   1:  PR[GP1:91,1] = PR[GP1:90,1] + -29.809;
   1:  PR[GP1:91,2] = PR[GP1:90,2] + -36.321;
   1:L PR[91] 10mm/sec CNT100;
   1:  PR[GP1:91,1] = PR[GP1:90,1] + -23.100;
   1:  PR[GP1:91,2] = PR[GP1:90,2] + -35.878;
   1:L PR[91] 10mm/sec CNT100;
   1:  PR[GP1:91,1] = PR[GP1:90,1] + -20.028;
   1:  PR[GP1:91,2] = PR[GP1:90,2] + -35.175;
   1:L PR[91] 10mm/sec CNT100;
   1:  PR[GP1:91,1] = PR[GP1:90,1] + -13.814;
   1:  PR[GP1:91,2] = PR[GP1:90,2] + -33.391;
   1:L PR[91] 10mm/sec CNT100;
   1:  PR[GP1:91,1] = PR[GP1:90,1] + -10.898;
   1:  PR[GP1:91,2] = PR[GP1:90,2] + -31.682;
   1:L PR[91] 10mm/sec CNT100;
   1:  PR[GP1:91,1] = PR[GP1:90,1] + -6.741;
   1:  PR[GP1:91,2] = PR[GP1:90,2] + -29.419;
   1:L PR[91] 10mm/sec CNT100;
   1:  PR[GP1:91,1] = PR[GP1:90,1] + -1.126;
   1:  PR[GP1:91,2] = PR[GP1:90,2] + -24.565;
   1:L PR[91] 10mm/sec CNT100;
   1:  PR[GP1:91,1] = PR[GP1:90,1] + -0.604;
   1:  PR[GP1:91,2] = PR[GP1:90,2] + -23.932;
   1:L PR[91] 10mm/sec CNT100;
   1:  PR[GP1:91,1] = PR[GP1:90,1] + 0.084;
   1:L PR[91] 10mm/sec CNT100;
   1:  PR[GP1:91,1] = PR[GP1:90,1] + 0.382;
   1:  PR[GP1:91,2] = PR[GP1:90,2] + -24.658;
   1:  PR[GP1:91,3] = PR[GP1:90,3] + 53.375;
   1:L PR[91] 10mm/sec CNT100;
   1:  PR[GP1:91,1] = PR[GP1:90,1] + 0.577;
   1:  PR[GP1:91,2] = PR[GP1:90,2] + -24.830;
   1:L PR[91] 10mm/sec CNT100;
   1:  PR[GP1:91,1] = PR[GP1:90,1] + 5.985;
   1:  PR[GP1:91,2] = PR[GP1:90,2] + -29.504;
   1:L PR[91] 10mm/sec CNT100;
   1:  PR[GP1:91,1] = PR[GP1:90,1] + 9.953;
   1:  PR[GP1:91,2] = PR[GP1:90,2] + -31.657;
   1:L PR[91] 10mm/sec CNT100;
   1:  PR[GP1:91,1] = PR[GP1:90,1] + 13.028;
   1:  PR[GP1:91,2] = PR[GP1:90,2] + -33.457;
   1:L PR[91] 10mm/sec CNT100;
   1:  PR[GP1:91,1] = PR[GP1:90,1] + 19.129;
   1:  PR[GP1:91,2] = PR[GP1:90,2] + -35.209;
   1:L PR[91] 10mm/sec CNT100;
   1:  PR[GP1:91,1] = PR[GP1:90,1] + 22.400;
   1:  PR[GP1:91,2] = PR[GP1:90,2] + -35.958;
   1:L PR[91] 10mm/sec CNT100;
   1:  PR[GP1:91,1] = PR[GP1:90,1] + 28.952;
   1:  PR[GP1:91,2] = PR[GP1:90,2] + -36.393;
   1:L PR[91] 10mm/sec CNT100;
   1:  PR[GP1:91,1] = PR[GP1:90,1] + 36.269;
   1:  PR[GP1:91,2] = PR[GP1:90,2] + -35.383;
   1:L PR[91] 10mm/sec CNT100;
   1:  PR[GP1:91,1] = PR[GP1:90,1] + 38.372;
   1:  PR[GP1:91,2] = PR[GP1:90,2] + -35.179;
   1:L PR[91] 10mm/sec CNT100;
   1:  PR[GP1:91,1] = PR[GP1:90,1] + 45.492;
   1:  PR[GP1:91,2] = PR[GP1:90,2] + -32.580;
   1:L PR[91] 10mm/sec CNT100;
   1:  PR[GP1:91,1] = PR[GP1:90,1] + 46.753;
   1:  PR[GP1:91,2] = PR[GP1:90,2] + -32.025;
   1:L PR[91] 10mm/sec CNT100;
   1:  PR[GP1:91,1] = PR[GP1:90,1] + 53.239;
   1:  PR[GP1:91,2] = PR[GP1:90,2] + -27.956;
   1:L PR[91] 10mm/sec CNT100;
   1:  PR[GP1:91,1] = PR[GP1:90,1] + 59.284;
   1:  PR[GP1:91,2] = PR[GP1:90,2] + -22.078;
   1:L PR[91] 10mm/sec CNT100;
   1:  PR[GP1:91,1] = PR[GP1:90,1] + 62.332;
   1:  PR[GP1:91,2] = PR[GP1:90,2] + -17.349;
   1:L PR[91] 10mm/sec CNT100;
   1:  PR[GP1:91,1] = PR[GP1:90,1] + 63.823;
   1:  PR[GP1:91,2] = PR[GP1:90,2] + -15.009;
   1:L PR[91] 10mm/sec CNT100;
   1:  PR[GP1:91,1] = PR[GP1:90,1] + 66.412;
   1:  PR[GP1:91,2] = PR[GP1:90,2] + -8.017;
   1:L PR[91] 10mm/sec CNT100;
   1:  PR[GP1:91,1] = PR[GP1:90,1] + 66.615;
   1:  PR[GP1:91,2] = PR[GP1:90,2] + -6.897;
   1:L PR[91] 10mm/sec CNT100;
   1:  PR[GP1:91,1] = PR[GP1:90,1] + 67.423;
   1:  PR[GP1:91,2] = PR[GP1:90,2] + 0.258;
   1:L PR[91] 10mm/sec CNT100;
   1:  PR[GP1:91,1] = PR[GP1:90,1] + 67.185;
   1:  PR[GP1:91,2] = PR[GP1:90,2] + 1.554;
   1:L PR[91] 10mm/sec CNT100;
   1:  PR[GP1:91,1] = PR[GP1:90,1] + 66.405;
   1:  PR[GP1:91,2] = PR[GP1:90,2] + 8.595;
   1:L PR[91] 10mm/sec CNT100;
   1:  PR[GP1:91,1] = PR[GP1:90,1] + 63.820;
   1:  PR[GP1:91,2] = PR[GP1:90,2] + 15.577;
   1:L PR[91] 10mm/sec CNT100;
   1:  PR[GP1:91,1] = PR[GP1:90,1] + 63.649;
   1:  PR[GP1:91,2] = PR[GP1:90,2] + 15.865;
   1:L PR[91] 10mm/sec CNT100;
   1:  PR[GP1:91,1] = PR[GP1:90,1] + 59.282;
   1:  PR[GP1:91,2] = PR[GP1:90,2] + 22.638;
   1:L PR[91] 10mm/sec CNT100;
   1:  PR[GP1:91,1] = PR[GP1:90,1] + 53.786;
   1:  PR[GP1:91,2] = PR[GP1:90,2] + 28.020;
   1:L PR[91] 10mm/sec CNT100;
   1:  PR[GP1:91,1] = PR[GP1:90,1] + 53.244;
   1:  PR[GP1:91,2] = PR[GP1:90,2] + 28.511;
   1:L PR[91] 10mm/sec CNT100;
   1:  PR[GP1:91,1] = PR[GP1:90,1] + 46.747;
   1:  PR[GP1:91,2] = PR[GP1:90,2] + 32.588;
   1:L PR[91] 10mm/sec CNT100;
   1:  PR[GP1:91,1] = PR[GP1:90,1] + 45.480;
   1:  PR[GP1:91,2] = PR[GP1:90,2] + 33.141;
   1:L PR[91] 10mm/sec CNT100;
   1:  PR[GP1:91,1] = PR[GP1:90,1] + 38.342;
   1:  PR[GP1:91,2] = PR[GP1:90,2] + 35.746;
   1:L PR[91] 10mm/sec CNT100;
   1:  PR[GP1:91,1] = PR[GP1:90,1] + 31.583;
   1:  PR[GP1:91,2] = PR[GP1:90,2] + 36.704;
   1:L PR[91] 10mm/sec CNT100;
   1:  PR[GP1:91,1] = PR[GP1:90,1] + 28.935;
   1:  PR[GP1:91,2] = PR[GP1:90,2] + 36.950;
   1:L PR[91] 10mm/sec CNT100;
   1:  PR[GP1:91,1] = PR[GP1:90,1] + 22.366;
   1:  PR[GP1:91,2] = PR[GP1:90,2] + 36.514;
   1:L PR[91] 10mm/sec CNT100;
   1:  PR[GP1:91,1] = PR[GP1:90,1] + 19.041;
   1:  PR[GP1:91,2] = PR[GP1:90,2] + 35.728;
   1:L PR[91] 10mm/sec CNT100;
   1:  PR[GP1:91,1] = PR[GP1:90,1] + 12.948;
   1:  PR[GP1:91,2] = PR[GP1:90,2] + 33.976;
   1:L PR[91] 10mm/sec CNT100;
   1:  PR[GP1:91,1] = PR[GP1:90,1] + 7.626;
   1:  PR[GP1:91,2] = PR[GP1:90,2] + 31.111;
   1:L PR[91] 10mm/sec CNT100;
   1:  PR[GP1:91,1] = PR[GP1:90,1] + 0.493;
   1:  PR[GP1:91,2] = PR[GP1:90,2] + 25.310;
   1:L PR[91] 10mm/sec CNT100;
   1:  PR[GP1:91,1] = PR[GP1:90,1] + 0.344;
   1:  PR[GP1:91,2] = PR[GP1:90,2] + 25.179;
   1:L PR[91] 10mm/sec CNT100;
   1:  PR[GP1:91,1] = PR[GP1:90,1] + 0.046;
   1:  PR[GP1:91,2] = PR[GP1:90,2] + 24.815;
   1:L PR[91] 10mm/sec CNT100;
   1:  PR[GP1:91,1] = PR[GP1:90,1] + -0.570;
   1:L PR[91] 10mm/sec CNT100;
   1:  PR[GP1:91,1] = PR[GP1:90,1] + -0.868;
   1:  PR[GP1:91,2] = PR[GP1:90,2] + 25.177;
   1:L PR[91] 10mm/sec CNT100;
   1:  PR[GP1:91,1] = PR[GP1:90,1] + -1.018;
   1:  PR[GP1:91,2] = PR[GP1:90,2] + 25.309;
   1:L PR[91] 10mm/sec CNT100;
   1:  PR[GP1:91,1] = PR[GP1:90,1] + -8.130;
   1:  PR[GP1:91,2] = PR[GP1:90,2] + 31.091;
   1:L PR[91] 10mm/sec CNT100;
   1:  PR[GP1:91,1] = PR[GP1:90,1] + -13.479;
   1:  PR[GP1:91,2] = PR[GP1:90,2] + 33.979;
   1:L PR[91] 10mm/sec CNT100;
   1:  PR[GP1:91,1] = PR[GP1:90,1] + -19.564;
   1:  PR[GP1:91,2] = PR[GP1:90,2] + 35.729;
   1:L PR[91] 10mm/sec CNT100;
   1:  PR[GP1:91,1] = PR[GP1:90,1] + -22.890;
   1:  PR[GP1:91,2] = PR[GP1:90,2] + 36.514;
   1:L PR[91] 10mm/sec CNT100;
   1:  PR[GP1:91,1] = PR[GP1:90,1] + -29.466;
   1:  PR[GP1:91,2] = PR[GP1:90,2] + 36.948;
   1:L PR[91] 10mm/sec CNT100;
   1:  PR[GP1:91,1] = PR[GP1:90,1] + -36.812;
   1:  PR[GP1:91,2] = PR[GP1:90,2] + 35.931;
   1:L PR[91] 10mm/sec CNT100;
   1:  PR[GP1:91,1] = PR[GP1:90,1] + -38.919;
   1:  PR[GP1:91,2] = PR[GP1:90,2] + 35.733;
   1:L PR[91] 10mm/sec CNT100;
   1:  PR[GP1:91,1] = PR[GP1:90,1] + -46.035;
   1:  PR[GP1:91,2] = PR[GP1:90,2] + 33.127;
   1:L PR[91] 10mm/sec CNT100;
   1:  PR[GP1:91,1] = PR[GP1:90,1] + -47.299;
   1:  PR[GP1:91,2] = PR[GP1:90,2] + 32.574;
   1:L PR[91] 10mm/sec CNT100;
   1:  PR[GP1:91,1] = PR[GP1:90,1] + -53.827;
   1:  PR[GP1:91,2] = PR[GP1:90,2] + 28.459;
   1:L PR[91] 10mm/sec CNT100;
   1:  PR[GP1:91,1] = PR[GP1:90,1] + -59.727;
   1:  PR[GP1:91,2] = PR[GP1:90,2] + 22.699;
   1:L PR[91] 10mm/sec CNT100;
   1:  PR[GP1:91,1] = PR[GP1:90,1] + -59.886;
   1:  PR[GP1:91,2] = PR[GP1:90,2] + 22.555;
   1:L PR[91] 10mm/sec CNT100;
   1:  PR[GP1:91,1] = PR[GP1:90,1] + -62.857;
   1:  PR[GP1:91,2] = PR[GP1:90,2] + 17.918;
   1:L PR[91] 10mm/sec CNT100;
   1:  PR[GP1:91,1] = PR[GP1:90,1] + -64.370;
   1:  PR[GP1:91,2] = PR[GP1:90,2] + 15.527;
   1:L PR[91] 10mm/sec CNT100;
   1:  PR[GP1:91,1] = PR[GP1:90,1] + -66.967;
   1:  PR[GP1:91,2] = PR[GP1:90,2] + 8.422;
   1:L PR[91] 10mm/sec CNT100;
   1:  PR[GP1:91,1] = PR[GP1:90,1] + -67.171;
   1:  PR[GP1:91,2] = PR[GP1:90,2] + 7.296;
   1:L PR[91] 10mm/sec CNT100;
   1:  PR[GP1:91,1] = PR[GP1:90,1] + -67.949;
   1:  PR[GP1:91,2] = PR[GP1:90,2] + 0.301;
   1:L PR[91] 10mm/sec CNT100;
   1:  PR[GP1:91,1] = PR[GP1:90,1] + -67.711;
   1:  PR[GP1:91,2] = PR[GP1:90,2] + -0.994;
   1:L PR[91] 10mm/sec CNT100;
   1:  PR[GP1:91,1] = PR[GP1:90,1] + -66.959;
   1:  PR[GP1:91,2] = PR[GP1:90,2] + -7.884;
   1:L PR[91] 10mm/sec CNT100;
   1:  PR[GP1:91,1] = PR[GP1:90,1] + -64.367;
   1:  PR[GP1:91,2] = PR[GP1:90,2] + -14.977;
   1:L PR[91] 10mm/sec CNT100;
   1:  PR[GP1:91,1] = PR[GP1:90,1] + -64.194;
   1:  PR[GP1:91,2] = PR[GP1:90,2] + -15.271;
   1:L PR[91] 10mm/sec CNT100;
   1:  PR[GP1:91,1] = PR[GP1:90,1] + -59.880;
   1:  PR[GP1:91,2] = PR[GP1:90,2] + -22.006;
   1:L PR[91] 10mm/sec CNT100;
   1:  PR[GP1:91,1] = PR[GP1:90,1] + -54.377;
   1:  PR[GP1:91,2] = PR[GP1:90,2] + -27.405;
   1:L PR[91] 10mm/sec CNT100;
   1:  PR[GP1:91,1] = PR[GP1:90,1] + -53.841;
   1:  PR[GP1:91,2] = PR[GP1:90,2] + -27.892;
   1:L PR[91] 10mm/sec CNT100;
   1:  PR[GP1:91,1] = PR[GP1:90,1] + -47.306;
   1:  PR[GP1:91,2] = PR[GP1:90,2] + -32.012;
   1:L PR[91] 10mm/sec CNT100;
   1:  PR[GP1:91,1] = PR[GP1:90,1] + -46.047;
   1:  PR[GP1:91,2] = PR[GP1:90,2] + -32.566;
   1:L PR[91] 10mm/sec CNT100;
   1:  PR[GP1:91,1] = PR[GP1:90,1] + -38.923;
   1:  PR[GP1:91,2] = PR[GP1:90,2] + -35.176;
   1:L PR[91] 10mm/sec CNT100;
   1:  PR[GP1:91,1] = PR[GP1:90,1] + -32.147;
   1:  PR[GP1:91,2] = PR[GP1:90,2] + -36.140;
   1:L PR[91] 10mm/sec CNT100;
   1:  PR[GP1:91,1] = PR[GP1:90,1] + -29.509;
   1:  PR[GP1:91,2] = PR[GP1:90,2] + -36.393;
   1:L PR[91] 10mm/sec CNT100;
   1:  PR[GP1:91,1] = PR[GP1:90,1] + -22.924;
   1:  PR[GP1:91,2] = PR[GP1:90,2] + -35.958;
   1:L PR[91] 10mm/sec CNT100;
   1:  PR[GP1:91,1] = PR[GP1:90,1] + -19.653;
   1:  PR[GP1:91,2] = PR[GP1:90,2] + -35.210;
   1:L PR[91] 10mm/sec CNT100;
   1:  PR[GP1:91,1] = PR[GP1:90,1] + -13.560;
   1:  PR[GP1:91,2] = PR[GP1:90,2] + -33.460;
   1:L PR[91] 10mm/sec CNT100;
   1:  PR[GP1:91,1] = PR[GP1:90,1] + -10.487;
   1:  PR[GP1:91,2] = PR[GP1:90,2] + -31.660;
   1:L PR[91] 10mm/sec CNT100;
   1:  PR[GP1:91,1] = PR[GP1:90,1] + -6.497;
   1:  PR[GP1:91,2] = PR[GP1:90,2] + -29.488;
   1:L PR[91] 10mm/sec CNT100;
   1:  PR[GP1:91,1] = PR[GP1:90,1] + -1.098;
   1:  PR[GP1:91,2] = PR[GP1:90,2] + -24.829;
   1:L PR[91] 10mm/sec CNT100;
   1:  PR[GP1:91,1] = PR[GP1:90,1] + -0.902;
   1:  PR[GP1:91,2] = PR[GP1:90,2] + -24.656;
   1:L PR[91] 10mm/sec CNT100;
   1:  PR[GP1:91,1] = PR[GP1:90,1] + -0.573;
   1:  PR[GP1:91,2] = PR[GP1:90,2] + -24.257;
   1:L PR[91] 10mm/sec CNT100;
   1:  PR[GP1:91,1] = PR[GP1:90,1] + 0.052;
   1:L PR[91] 10mm/sec CNT100;
   1:  PR[GP1:91,1] = PR[GP1:90,1] + 5.741;
   1:  PR[GP1:91,2] = PR[GP1:90,2] + -29.572;
   1:  PR[GP1:91,3] = PR[GP1:90,3] + 53.985;
   1:L PR[91] 10mm/sec CNT100;
   1:  PR[GP1:91,1] = PR[GP1:90,1] + 9.542;
   1:  PR[GP1:91,2] = PR[GP1:90,2] + -31.635;
   1:L PR[91] 10mm/sec CNT100;
   1:  PR[GP1:91,1] = PR[GP1:90,1] + 12.773;
   1:  PR[GP1:91,2] = PR[GP1:90,2] + -33.526;
   1:L PR[91] 10mm/sec CNT100;
   1:  PR[GP1:91,1] = PR[GP1:90,1] + 18.753;
   1:  PR[GP1:91,2] = PR[GP1:90,2] + -35.244;
   1:L PR[91] 10mm/sec CNT100;
   1:  PR[GP1:91,1] = PR[GP1:90,1] + 22.223;
   1:  PR[GP1:91,2] = PR[GP1:90,2] + -36.038;
   1:L PR[91] 10mm/sec CNT100;
   1:  PR[GP1:91,1] = PR[GP1:90,1] + 28.652;
   1:  PR[GP1:91,2] = PR[GP1:90,2] + -36.465;
   1:L PR[91] 10mm/sec CNT100;
   1:  PR[GP1:91,1] = PR[GP1:90,1] + 35.832;
   1:  PR[GP1:91,2] = PR[GP1:90,2] + -35.474;
   1:L PR[91] 10mm/sec CNT100;
   1:  PR[GP1:91,1] = PR[GP1:90,1] + 38.154;
   1:  PR[GP1:91,2] = PR[GP1:90,2] + -35.248;
   1:L PR[91] 10mm/sec CNT100;
   1:  PR[GP1:91,1] = PR[GP1:90,1] + 45.148;
   1:  PR[GP1:91,2] = PR[GP1:90,2] + -32.696;
   1:L PR[91] 10mm/sec CNT100;
   1:  PR[GP1:91,1] = PR[GP1:90,1] + 46.608;
   1:  PR[GP1:91,2] = PR[GP1:90,2] + -32.053;
   1:L PR[91] 10mm/sec CNT100;
   1:  PR[GP1:91,1] = PR[GP1:90,1] + 52.984;
   1:  PR[GP1:91,2] = PR[GP1:90,2] + -28.053;
   1:L PR[91] 10mm/sec CNT100;
   1:  PR[GP1:91,1] = PR[GP1:90,1] + 58.770;
   1:  PR[GP1:91,2] = PR[GP1:90,2] + -22.413;
   1:L PR[91] 10mm/sec CNT100;
   1:  PR[GP1:91,1] = PR[GP1:90,1] + 59.102;
   1:  PR[GP1:91,2] = PR[GP1:90,2] + -22.111;
   1:L PR[91] 10mm/sec CNT100;
   1:  PR[GP1:91,1] = PR[GP1:90,1] + 63.606;
   1:  PR[GP1:91,2] = PR[GP1:90,2] + -15.115;
   1:L PR[91] 10mm/sec CNT100;
   1:  PR[GP1:91,1] = PR[GP1:90,1] + 66.309;
   1:  PR[GP1:91,2] = PR[GP1:90,2] + -7.800;
   1:L PR[91] 10mm/sec CNT100;
   1:  PR[GP1:91,1] = PR[GP1:90,1] + 66.390;
   1:  PR[GP1:91,2] = PR[GP1:90,2] + -7.350;
   1:L PR[91] 10mm/sec CNT100;
   1:  PR[GP1:91,1] = PR[GP1:90,1] + 67.249;
   1:  PR[GP1:91,2] = PR[GP1:90,2] + 0.258;
   1:L PR[91] 10mm/sec CNT100;
   1:  PR[GP1:91,1] = PR[GP1:90,1] + 67.127;
   1:  PR[GP1:91,2] = PR[GP1:90,2] + 0.921;
   1:L PR[91] 10mm/sec CNT100;
   1:  PR[GP1:91,1] = PR[GP1:90,1] + 66.301;
   1:  PR[GP1:91,2] = PR[GP1:90,2] + 8.377;
   1:L PR[91] 10mm/sec CNT100;
   1:  PR[GP1:91,1] = PR[GP1:90,1] + 63.606;
   1:  PR[GP1:91,2] = PR[GP1:90,2] + 15.673;
   1:L PR[91] 10mm/sec CNT100;
   1:  PR[GP1:91,1] = PR[GP1:90,1] + 59.095;
   1:  PR[GP1:91,2] = PR[GP1:90,2] + 22.680;
   1:L PR[91] 10mm/sec CNT100;
   1:  PR[GP1:91,1] = PR[GP1:90,1] + 53.689;
   1:  PR[GP1:91,2] = PR[GP1:90,2] + 27.974;
   1:L PR[91] 10mm/sec CNT100;
   1:  PR[GP1:91,1] = PR[GP1:90,1] + 52.987;
   1:  PR[GP1:91,2] = PR[GP1:90,2] + 28.609;
   1:L PR[91] 10mm/sec CNT100;
   1:  PR[GP1:91,1] = PR[GP1:90,1] + 46.600;
   1:  PR[GP1:91,2] = PR[GP1:90,2] + 32.617;
   1:L PR[91] 10mm/sec CNT100;
   1:  PR[GP1:91,1] = PR[GP1:90,1] + 45.134;
   1:  PR[GP1:91,2] = PR[GP1:90,2] + 33.257;
   1:L PR[91] 10mm/sec CNT100;
   1:  PR[GP1:91,1] = PR[GP1:90,1] + 38.123;
   1:  PR[GP1:91,2] = PR[GP1:90,2] + 35.816;
   1:L PR[91] 10mm/sec CNT100;
   1:  PR[GP1:91,1] = PR[GP1:90,1] + 31.484;
   1:  PR[GP1:91,2] = PR[GP1:90,2] + 36.757;
   1:L PR[91] 10mm/sec CNT100;
   1:  PR[GP1:91,1] = PR[GP1:90,1] + 28.633;
   1:  PR[GP1:91,2] = PR[GP1:90,2] + 37.022;
   1:L PR[91] 10mm/sec CNT100;
   1:  PR[GP1:91,1] = PR[GP1:90,1] + 22.187;
   1:  PR[GP1:91,2] = PR[GP1:90,2] + 36.594;
   1:L PR[91] 10mm/sec CNT100;
   1:  PR[GP1:91,1] = PR[GP1:90,1] + 18.660;
   1:  PR[GP1:91,2] = PR[GP1:90,2] + 35.761;
   1:L PR[91] 10mm/sec CNT100;
   1:  PR[GP1:91,1] = PR[GP1:90,1] + 12.690;
   1:  PR[GP1:91,2] = PR[GP1:90,2] + 34.044;
   1:L PR[91] 10mm/sec CNT100;
   1:  PR[GP1:91,1] = PR[GP1:90,1] + 7.453;
   1:  PR[GP1:91,2] = PR[GP1:90,2] + 31.225;
   1:L PR[91] 10mm/sec CNT100;
   1:  PR[GP1:91,1] = PR[GP1:90,1] + -0.263;
   1:  PR[GP1:91,2] = PR[GP1:90,2] + 24.950;
   1:L PR[91] 10mm/sec CNT100;
   1:  PR[GP1:91,1] = PR[GP1:90,1] + -7.958;
   1:  PR[GP1:91,2] = PR[GP1:90,2] + 31.206;
   1:L PR[91] 10mm/sec CNT100;
   1:  PR[GP1:91,1] = PR[GP1:90,1] + -13.221;
   1:  PR[GP1:91,2] = PR[GP1:90,2] + 34.047;
   1:L PR[91] 10mm/sec CNT100;
   1:  PR[GP1:91,1] = PR[GP1:90,1] + -19.183;
   1:  PR[GP1:91,2] = PR[GP1:90,2] + 35.761;
   1:L PR[91] 10mm/sec CNT100;
   1:  PR[GP1:91,1] = PR[GP1:90,1] + -22.711;
   1:  PR[GP1:91,2] = PR[GP1:90,2] + 36.594;
   1:L PR[91] 10mm/sec CNT100;
   1:  PR[GP1:91,1] = PR[GP1:90,1] + -29.163;
   1:  PR[GP1:91,2] = PR[GP1:90,2] + 37.020;
   1:L PR[91] 10mm/sec CNT100;
   1:  PR[GP1:91,1] = PR[GP1:90,1] + -36.373;
   1:  PR[GP1:91,2] = PR[GP1:90,2] + 36.022;
   1:L PR[91] 10mm/sec CNT100;
   1:  PR[GP1:91,1] = PR[GP1:90,1] + -38.699;
   1:  PR[GP1:91,2] = PR[GP1:90,2] + 35.803;
   1:L PR[91] 10mm/sec CNT100;
   1:  PR[GP1:91,1] = PR[GP1:90,1] + -45.689;
   1:  PR[GP1:91,2] = PR[GP1:90,2] + 33.243;
   1:L PR[91] 10mm/sec CNT100;
   1:  PR[GP1:91,1] = PR[GP1:90,1] + -47.153;
   1:  PR[GP1:91,2] = PR[GP1:90,2] + 32.603;
   1:L PR[91] 10mm/sec CNT100;
   1:  PR[GP1:91,1] = PR[GP1:90,1] + -53.569;
   1:  PR[GP1:91,2] = PR[GP1:90,2] + 28.558;
   1:L PR[91] 10mm/sec CNT100;
   1:  PR[GP1:91,1] = PR[GP1:90,1] + -59.370;
   1:  PR[GP1:91,2] = PR[GP1:90,2] + 22.895;
   1:L PR[91] 10mm/sec CNT100;
   1:  PR[GP1:91,1] = PR[GP1:90,1] + -59.698;
   1:  PR[GP1:91,2] = PR[GP1:90,2] + 22.598;
   1:L PR[91] 10mm/sec CNT100;
   1:  PR[GP1:91,1] = PR[GP1:90,1] + -64.153;
   1:  PR[GP1:91,2] = PR[GP1:90,2] + 15.634;
   1:L PR[91] 10mm/sec CNT100;
   1:  PR[GP1:91,1] = PR[GP1:90,1] + -66.865;
   1:  PR[GP1:91,2] = PR[GP1:90,2] + 8.197;
   1:L PR[91] 10mm/sec CNT100;
   1:  PR[GP1:91,1] = PR[GP1:90,1] + -66.948;
   1:  PR[GP1:91,2] = PR[GP1:90,2] + 7.740;
   1:L PR[91] 10mm/sec CNT100;
   1:  PR[GP1:91,1] = PR[GP1:90,1] + -67.775;
   1:  PR[GP1:91,2] = PR[GP1:90,2] + 0.301;
   1:L PR[91] 10mm/sec CNT100;
   1:  PR[GP1:91,1] = PR[GP1:90,1] + -67.653;
   1:  PR[GP1:91,2] = PR[GP1:90,2] + -0.362;
   1:L PR[91] 10mm/sec CNT100;
   1:  PR[GP1:91,1] = PR[GP1:90,1] + -66.857;
   1:  PR[GP1:91,2] = PR[GP1:90,2] + -7.659;
   1:L PR[91] 10mm/sec CNT100;
   1:  PR[GP1:91,1] = PR[GP1:90,1] + -64.146;
   1:  PR[GP1:91,2] = PR[GP1:90,2] + -15.094;
   1:L PR[91] 10mm/sec CNT100;
   1:  PR[GP1:91,1] = PR[GP1:90,1] + -64.138;
   1:  PR[GP1:91,2] = PR[GP1:90,2] + -15.110;
   1:L PR[91] 10mm/sec CNT100;
   1:  PR[GP1:91,1] = PR[GP1:90,1] + -59.692;
   1:  PR[GP1:91,2] = PR[GP1:90,2] + -22.049;
   1:L PR[91] 10mm/sec CNT100;
   1:  PR[GP1:91,1] = PR[GP1:90,1] + -54.279;
   1:  PR[GP1:91,2] = PR[GP1:90,2] + -27.360;
   1:L PR[91] 10mm/sec CNT100;
   1:  PR[GP1:91,1] = PR[GP1:90,1] + -53.584;
   1:  PR[GP1:91,2] = PR[GP1:90,2] + -27.990;
   1:L PR[91] 10mm/sec CNT100;
   1:  PR[GP1:91,1] = PR[GP1:90,1] + -47.161;
   1:  PR[GP1:91,2] = PR[GP1:90,2] + -32.040;
   1:L PR[91] 10mm/sec CNT100;
   1:  PR[GP1:91,1] = PR[GP1:90,1] + -45.703;
   1:  PR[GP1:91,2] = PR[GP1:90,2] + -32.682;
   1:L PR[91] 10mm/sec CNT100;
   1:  PR[GP1:91,1] = PR[GP1:90,1] + -38.705;
   1:  PR[GP1:91,2] = PR[GP1:90,2] + -35.245;
   1:L PR[91] 10mm/sec CNT100;
   1:  PR[GP1:91,1] = PR[GP1:90,1] + -32.049;
   1:  PR[GP1:91,2] = PR[GP1:90,2] + -36.192;
   1:L PR[91] 10mm/sec CNT100;
   1:  PR[GP1:91,1] = PR[GP1:90,1] + -29.209;
   1:  PR[GP1:91,2] = PR[GP1:90,2] + -36.465;
   1:L PR[91] 10mm/sec CNT100;
   1:  PR[GP1:91,1] = PR[GP1:90,1] + -22.747;
   1:  PR[GP1:91,2] = PR[GP1:90,2] + -36.038;
   1:L PR[91] 10mm/sec CNT100;
   1:  PR[GP1:91,1] = PR[GP1:90,1] + -19.277;
   1:  PR[GP1:91,2] = PR[GP1:90,2] + -35.245;
   1:L PR[91] 10mm/sec CNT100;
   1:  PR[GP1:91,1] = PR[GP1:90,1] + -13.305;
   1:  PR[GP1:91,2] = PR[GP1:90,2] + -33.529;
   1:L PR[91] 10mm/sec CNT100;
   1:  PR[GP1:91,1] = PR[GP1:90,1] + -10.076;
   1:  PR[GP1:91,2] = PR[GP1:90,2] + -31.638;
   1:L PR[91] 10mm/sec CNT100;
   1:  PR[GP1:91,1] = PR[GP1:90,1] + -6.254;
   1:  PR[GP1:91,2] = PR[GP1:90,2] + -29.557;
   1:L PR[91] 10mm/sec CNT100;
   1:  PR[GP1:91,1] = PR[GP1:90,1] + -0.261;
   1:  PR[GP1:91,2] = PR[GP1:90,2] + -24.385;
   1:L PR[91] 10mm/sec CNT100;
   1:  PR[GP1:91,1] = PR[GP1:90,1] + 5.496;
   1:  PR[GP1:91,2] = PR[GP1:90,2] + -29.641;
   1:  PR[GP1:91,3] = PR[GP1:90,3] + 54.595;
   1:L PR[91] 10mm/sec CNT100;
   1:  PR[GP1:91,1] = PR[GP1:90,1] + 9.132;
   1:  PR[GP1:91,2] = PR[GP1:90,2] + -31.614;
   1:L PR[91] 10mm/sec CNT100;
   1:  PR[GP1:91,1] = PR[GP1:90,1] + 12.518;
   1:  PR[GP1:91,2] = PR[GP1:90,2] + -33.596;
   1:L PR[91] 10mm/sec CNT100;
   1:  PR[GP1:91,1] = PR[GP1:90,1] + 18.378;
   1:  PR[GP1:91,2] = PR[GP1:90,2] + -35.279;
   1:L PR[91] 10mm/sec CNT100;
   1:  PR[GP1:91,1] = PR[GP1:90,1] + 22.046;
   1:  PR[GP1:91,2] = PR[GP1:90,2] + -36.118;
   1:L PR[91] 10mm/sec CNT100;
   1:  PR[GP1:91,1] = PR[GP1:90,1] + 28.352;
   1:  PR[GP1:91,2] = PR[GP1:90,2] + -36.537;
   1:L PR[91] 10mm/sec CNT100;
   1:  PR[GP1:91,1] = PR[GP1:90,1] + 35.396;
   1:  PR[GP1:91,2] = PR[GP1:90,2] + -35.565;
   1:L PR[91] 10mm/sec CNT100;
   1:  PR[GP1:91,1] = PR[GP1:90,1] + 37.937;
   1:  PR[GP1:91,2] = PR[GP1:90,2] + -35.318;
   1:L PR[91] 10mm/sec CNT100;
   1:  PR[GP1:91,1] = PR[GP1:90,1] + 44.804;
   1:  PR[GP1:91,2] = PR[GP1:90,2] + -32.811;
   1:L PR[91] 10mm/sec CNT100;
   1:  PR[GP1:91,1] = PR[GP1:90,1] + 46.463;
   1:  PR[GP1:91,2] = PR[GP1:90,2] + -32.082;
   1:L PR[91] 10mm/sec CNT100;
   1:  PR[GP1:91,1] = PR[GP1:90,1] + 52.728;
   1:  PR[GP1:91,2] = PR[GP1:90,2] + -28.151;
   1:L PR[91] 10mm/sec CNT100;
   1:  PR[GP1:91,1] = PR[GP1:90,1] + 58.415;
   1:  PR[GP1:91,2] = PR[GP1:90,2] + -22.607;
   1:L PR[91] 10mm/sec CNT100;
   1:  PR[GP1:91,1] = PR[GP1:90,1] + 58.915;
   1:  PR[GP1:91,2] = PR[GP1:90,2] + -22.153;
   1:L PR[91] 10mm/sec CNT100;
   1:  PR[GP1:91,1] = PR[GP1:90,1] + 63.327;
   1:  PR[GP1:91,2] = PR[GP1:90,2] + -15.309;
   1:L PR[91] 10mm/sec CNT100;
   1:  PR[GP1:91,1] = PR[GP1:90,1] + 63.445;
   1:  PR[GP1:91,2] = PR[GP1:90,2] + -15.097;
   1:L PR[91] 10mm/sec CNT100;
   1:  PR[GP1:91,1] = PR[GP1:90,1] + 66.176;
   1:  PR[GP1:91,2] = PR[GP1:90,2] + -7.670;
   1:L PR[91] 10mm/sec CNT100;
   1:  PR[GP1:91,1] = PR[GP1:90,1] + 67.077;
   1:  PR[GP1:91,2] = PR[GP1:90,2] + 0.279;
   1:L PR[91] 10mm/sec CNT100;
   1:  PR[GP1:91,1] = PR[GP1:90,1] + 66.176;
   1:  PR[GP1:91,2] = PR[GP1:90,2] + 8.228;
   1:L PR[91] 10mm/sec CNT100;
   1:  PR[GP1:91,1] = PR[GP1:90,1] + 63.445;
   1:  PR[GP1:91,2] = PR[GP1:90,2] + 15.656;
   1:L PR[91] 10mm/sec CNT100;
   1:  PR[GP1:91,1] = PR[GP1:90,1] + 63.327;
   1:  PR[GP1:91,2] = PR[GP1:90,2] + 15.868;
   1:L PR[91] 10mm/sec CNT100;
   1:  PR[GP1:91,1] = PR[GP1:90,1] + 58.907;
   1:  PR[GP1:91,2] = PR[GP1:90,2] + 22.722;
   1:L PR[91] 10mm/sec CNT100;
   1:  PR[GP1:91,1] = PR[GP1:90,1] + 53.591;
   1:  PR[GP1:91,2] = PR[GP1:90,2] + 27.928;
   1:L PR[91] 10mm/sec CNT100;
   1:  PR[GP1:91,1] = PR[GP1:90,1] + 52.731;
   1:  PR[GP1:91,2] = PR[GP1:90,2] + 28.707;
   1:L PR[91] 10mm/sec CNT100;
   1:  PR[GP1:91,1] = PR[GP1:90,1] + 46.454;
   1:  PR[GP1:91,2] = PR[GP1:90,2] + 32.646;
   1:L PR[91] 10mm/sec CNT100;
   1:  PR[GP1:91,1] = PR[GP1:90,1] + 44.788;
   1:  PR[GP1:91,2] = PR[GP1:90,2] + 33.373;
   1:L PR[91] 10mm/sec CNT100;
   1:  PR[GP1:91,1] = PR[GP1:90,1] + 37.903;
   1:  PR[GP1:91,2] = PR[GP1:90,2] + 35.886;
   1:L PR[91] 10mm/sec CNT100;
   1:  PR[GP1:91,1] = PR[GP1:90,1] + 31.385;
   1:  PR[GP1:91,2] = PR[GP1:90,2] + 36.810;
   1:L PR[91] 10mm/sec CNT100;
   1:  PR[GP1:91,1] = PR[GP1:90,1] + 28.331;
   1:  PR[GP1:91,2] = PR[GP1:90,2] + 37.094;
   1:L PR[91] 10mm/sec CNT100;
   1:  PR[GP1:91,1] = PR[GP1:90,1] + 22.009;
   1:  PR[GP1:91,2] = PR[GP1:90,2] + 36.674;
   1:L PR[91] 10mm/sec CNT100;
   1:  PR[GP1:91,1] = PR[GP1:90,1] + 18.280;
   1:  PR[GP1:91,2] = PR[GP1:90,2] + 35.793;
   1:L PR[91] 10mm/sec CNT100;
   1:  PR[GP1:91,1] = PR[GP1:90,1] + 12.432;
   1:  PR[GP1:91,2] = PR[GP1:90,2] + 34.112;
   1:L PR[91] 10mm/sec CNT100;
   1:  PR[GP1:91,1] = PR[GP1:90,1] + 7.280;
   1:  PR[GP1:91,2] = PR[GP1:90,2] + 31.339;
   1:L PR[91] 10mm/sec CNT100;
   1:  PR[GP1:91,1] = PR[GP1:90,1] + -0.263;
   1:  PR[GP1:91,2] = PR[GP1:90,2] + 25.204;
   1:L PR[91] 10mm/sec CNT100;
   1:  PR[GP1:91,1] = PR[GP1:90,1] + -7.786;
   1:  PR[GP1:91,2] = PR[GP1:90,2] + 31.321;
   1:L PR[91] 10mm/sec CNT100;
   1:  PR[GP1:91,1] = PR[GP1:90,1] + -12.962;
   1:  PR[GP1:91,2] = PR[GP1:90,2] + 34.115;
   1:L PR[91] 10mm/sec CNT100;
   1:  PR[GP1:91,1] = PR[GP1:90,1] + -18.802;
   1:  PR[GP1:91,2] = PR[GP1:90,2] + 35.794;
   1:L PR[91] 10mm/sec CNT100;
   1:  PR[GP1:91,1] = PR[GP1:90,1] + -22.532;
   1:  PR[GP1:91,2] = PR[GP1:90,2] + 36.674;
   1:L PR[91] 10mm/sec CNT100;
   1:  PR[GP1:91,1] = PR[GP1:90,1] + -28.861;
   1:  PR[GP1:91,2] = PR[GP1:90,2] + 37.092;
   1:L PR[91] 10mm/sec CNT100;
   1:  PR[GP1:91,1] = PR[GP1:90,1] + -35.934;
   1:  PR[GP1:91,2] = PR[GP1:90,2] + 36.113;
   1:L PR[91] 10mm/sec CNT100;
   1:  PR[GP1:91,1] = PR[GP1:90,1] + -38.479;
   1:  PR[GP1:91,2] = PR[GP1:90,2] + 35.874;
   1:L PR[91] 10mm/sec CNT100;
   1:  PR[GP1:91,1] = PR[GP1:90,1] + -45.342;
   1:  PR[GP1:91,2] = PR[GP1:90,2] + 33.360;
   1:L PR[91] 10mm/sec CNT100;
   1:  PR[GP1:91,1] = PR[GP1:90,1] + -47.006;
   1:  PR[GP1:91,2] = PR[GP1:90,2] + 32.633;
   1:L PR[91] 10mm/sec CNT100;
   1:  PR[GP1:91,1] = PR[GP1:90,1] + -53.311;
   1:  PR[GP1:91,2] = PR[GP1:90,2] + 28.657;
   1:L PR[91] 10mm/sec CNT100;
   1:  PR[GP1:91,1] = PR[GP1:90,1] + -59.012;
   1:  PR[GP1:91,2] = PR[GP1:90,2] + 23.092;
   1:L PR[91] 10mm/sec CNT100;
   1:  PR[GP1:91,1] = PR[GP1:90,1] + -59.509;
   1:  PR[GP1:91,2] = PR[GP1:90,2] + 22.642;
   1:L PR[91] 10mm/sec CNT100;
   1:  PR[GP1:91,1] = PR[GP1:90,1] + -63.875;
   1:  PR[GP1:91,2] = PR[GP1:90,2] + 15.828;
   1:L PR[91] 10mm/sec CNT100;
   1:  PR[GP1:91,1] = PR[GP1:90,1] + -63.992;
   1:  PR[GP1:91,2] = PR[GP1:90,2] + 15.617;
   1:L PR[91] 10mm/sec CNT100;
   1:  PR[GP1:91,1] = PR[GP1:90,1] + -66.735;
   1:  PR[GP1:91,2] = PR[GP1:90,2] + 8.058;
   1:L PR[91] 10mm/sec CNT100;
   1:  PR[GP1:91,1] = PR[GP1:90,1] + -67.601;
   1:  PR[GP1:91,2] = PR[GP1:90,2] + 0.301;
   1:L PR[91] 10mm/sec CNT100;
   1:  PR[GP1:91,1] = PR[GP1:90,1] + -67.596;
   1:  PR[GP1:91,2] = PR[GP1:90,2] + 0.270;
   1:L PR[91] 10mm/sec CNT100;
   1:  PR[GP1:91,1] = PR[GP1:90,1] + -66.735;
   1:  PR[GP1:91,2] = PR[GP1:90,2] + -7.500;
   1:L PR[91] 10mm/sec CNT100;
   1:  PR[GP1:91,1] = PR[GP1:90,1] + -63.992;
   1:  PR[GP1:91,2] = PR[GP1:90,2] + -15.058;
   1:L PR[91] 10mm/sec CNT100;
   1:  PR[GP1:91,1] = PR[GP1:90,1] + -63.876;
   1:  PR[GP1:91,2] = PR[GP1:90,2] + -15.269;
   1:L PR[91] 10mm/sec CNT100;
   1:  PR[GP1:91,1] = PR[GP1:90,1] + -59.504;
   1:  PR[GP1:91,2] = PR[GP1:90,2] + -22.092;
   1:L PR[91] 10mm/sec CNT100;
   1:  PR[GP1:91,1] = PR[GP1:90,1] + -54.181;
   1:  PR[GP1:91,2] = PR[GP1:90,2] + -27.314;
   1:L PR[91] 10mm/sec CNT100;
   1:  PR[GP1:91,1] = PR[GP1:90,1] + -53.327;
   1:  PR[GP1:91,2] = PR[GP1:90,2] + -28.089;
   1:L PR[91] 10mm/sec CNT100;
   1:  PR[GP1:91,1] = PR[GP1:90,1] + -47.015;
   1:  PR[GP1:91,2] = PR[GP1:90,2] + -32.069;
   1:L PR[91] 10mm/sec CNT100;
   1:  PR[GP1:91,1] = PR[GP1:90,1] + -45.358;
   1:  PR[GP1:91,2] = PR[GP1:90,2] + -32.798;
   1:L PR[91] 10mm/sec CNT100;
   1:  PR[GP1:91,1] = PR[GP1:90,1] + -38.487;
   1:  PR[GP1:91,2] = PR[GP1:90,2] + -35.315;
   1:L PR[91] 10mm/sec CNT100;
   1:  PR[GP1:91,1] = PR[GP1:90,1] + -31.951;
   1:  PR[GP1:91,2] = PR[GP1:90,2] + -36.245;
   1:L PR[91] 10mm/sec CNT100;
   1:  PR[GP1:91,1] = PR[GP1:90,1] + -28.908;
   1:  PR[GP1:91,2] = PR[GP1:90,2] + -36.537;
   1:L PR[91] 10mm/sec CNT100;
   1:  PR[GP1:91,1] = PR[GP1:90,1] + -22.570;
   1:  PR[GP1:91,2] = PR[GP1:90,2] + -36.118;
   1:L PR[91] 10mm/sec CNT100;
   1:  PR[GP1:91,1] = PR[GP1:90,1] + -18.902;
   1:  PR[GP1:91,2] = PR[GP1:90,2] + -35.279;
   1:L PR[91] 10mm/sec CNT100;
   1:  PR[GP1:91,1] = PR[GP1:90,1] + -13.050;
   1:  PR[GP1:91,2] = PR[GP1:90,2] + -33.599;
   1:L PR[91] 10mm/sec CNT100;
   1:  PR[GP1:91,1] = PR[GP1:90,1] + -9.666;
   1:  PR[GP1:91,2] = PR[GP1:90,2] + -31.616;
   1:L PR[91] 10mm/sec CNT100;
   1:  PR[GP1:91,1] = PR[GP1:90,1] + -6.010;
   1:  PR[GP1:91,2] = PR[GP1:90,2] + -29.626;
   1:L PR[91] 10mm/sec CNT100;
   1:  PR[GP1:91,1] = PR[GP1:90,1] + -0.261;
   1:  PR[GP1:91,2] = PR[GP1:90,2] + -24.665;
   1:L PR[91] 10mm/sec CNT100;
   1:  PR[GP1:91,1] = PR[GP1:90,1] + 5.252;
   1:  PR[GP1:91,2] = PR[GP1:90,2] + -29.709;
   1:  PR[GP1:91,3] = PR[GP1:90,3] + 55.205;
   1:L PR[91] 10mm/sec CNT100;
   1:  PR[GP1:91,1] = PR[GP1:90,1] + 8.721;
   1:  PR[GP1:91,2] = PR[GP1:90,2] + -31.592;
   1:L PR[91] 10mm/sec CNT100;
   1:  PR[GP1:91,1] = PR[GP1:90,1] + 12.264;
   1:  PR[GP1:91,2] = PR[GP1:90,2] + -33.665;
   1:L PR[91] 10mm/sec CNT100;
   1:  PR[GP1:91,1] = PR[GP1:90,1] + 18.003;
   1:  PR[GP1:91,2] = PR[GP1:90,2] + -35.314;
   1:L PR[91] 10mm/sec CNT100;
   1:  PR[GP1:91,1] = PR[GP1:90,1] + 21.869;
   1:  PR[GP1:91,2] = PR[GP1:90,2] + -36.198;
   1:L PR[91] 10mm/sec CNT100;
   1:  PR[GP1:91,1] = PR[GP1:90,1] + 28.052;
   1:  PR[GP1:91,2] = PR[GP1:90,2] + -36.609;
   1:L PR[91] 10mm/sec CNT100;
   1:  PR[GP1:91,1] = PR[GP1:90,1] + 34.960;
   1:  PR[GP1:91,2] = PR[GP1:90,2] + -35.655;
   1:L PR[91] 10mm/sec CNT100;
   1:  PR[GP1:91,1] = PR[GP1:90,1] + 37.719;
   1:  PR[GP1:91,2] = PR[GP1:90,2] + -35.387;
   1:L PR[91] 10mm/sec CNT100;
   1:  PR[GP1:91,1] = PR[GP1:90,1] + 44.460;
   1:  PR[GP1:91,2] = PR[GP1:90,2] + -32.927;
   1:L PR[91] 10mm/sec CNT100;
   1:  PR[GP1:91,1] = PR[GP1:90,1] + 46.318;
   1:  PR[GP1:91,2] = PR[GP1:90,2] + -32.110;
   1:L PR[91] 10mm/sec CNT100;
   1:  PR[GP1:91,1] = PR[GP1:90,1] + 52.472;
   1:  PR[GP1:91,2] = PR[GP1:90,2] + -28.248;
   1:L PR[91] 10mm/sec CNT100;
   1:  PR[GP1:91,1] = PR[GP1:90,1] + 58.060;
   1:  PR[GP1:91,2] = PR[GP1:90,2] + -22.802;
   1:L PR[91] 10mm/sec CNT100;
   1:  PR[GP1:91,1] = PR[GP1:90,1] + 58.728;
   1:  PR[GP1:91,2] = PR[GP1:90,2] + -22.194;
   1:L PR[91] 10mm/sec CNT100;
   1:  PR[GP1:91,1] = PR[GP1:90,1] + 63.066;
   1:  PR[GP1:91,2] = PR[GP1:90,2] + -15.467;
   1:L PR[91] 10mm/sec CNT100;
   1:  PR[GP1:91,1] = PR[GP1:90,1] + 63.290;
   1:  PR[GP1:91,2] = PR[GP1:90,2] + -15.061;
   1:L PR[91] 10mm/sec CNT100;
   1:  PR[GP1:91,1] = PR[GP1:90,1] + 65.977;
   1:  PR[GP1:91,2] = PR[GP1:90,2] + -7.756;
   1:L PR[91] 10mm/sec CNT100;
   1:  PR[GP1:91,1] = PR[GP1:90,1] + 66.879;
   1:  PR[GP1:91,2] = PR[GP1:90,2] + 0.177;
   1:L PR[91] 10mm/sec CNT100;
   1:  PR[GP1:91,1] = PR[GP1:90,1] + 66.899;
   1:  PR[GP1:91,2] = PR[GP1:90,2] + 0.296;
   1:L PR[91] 10mm/sec CNT100;
   1:  PR[GP1:91,1] = PR[GP1:90,1] + 66.016;
   1:  PR[GP1:91,2] = PR[GP1:90,2] + 8.103;
   1:L PR[91] 10mm/sec CNT100;
   1:  PR[GP1:91,1] = PR[GP1:90,1] + 65.983;
   1:  PR[GP1:91,2] = PR[GP1:90,2] + 8.299;
   1:L PR[91] 10mm/sec CNT100;
   1:  PR[GP1:91,1] = PR[GP1:90,1] + 63.290;
   1:  PR[GP1:91,2] = PR[GP1:90,2] + 15.619;
   1:L PR[91] 10mm/sec CNT100;
   1:  PR[GP1:91,1] = PR[GP1:90,1] + 63.064;
   1:  PR[GP1:91,2] = PR[GP1:90,2] + 16.027;
   1:L PR[91] 10mm/sec CNT100;
   1:  PR[GP1:91,1] = PR[GP1:90,1] + 58.720;
   1:  PR[GP1:91,2] = PR[GP1:90,2] + 22.765;
   1:L PR[91] 10mm/sec CNT100;
   1:  PR[GP1:91,1] = PR[GP1:90,1] + 53.494;
   1:  PR[GP1:91,2] = PR[GP1:90,2] + 27.882;
   1:L PR[91] 10mm/sec CNT100;
   1:  PR[GP1:91,1] = PR[GP1:90,1] + 52.474;
   1:  PR[GP1:91,2] = PR[GP1:90,2] + 28.806;
   1:L PR[91] 10mm/sec CNT100;
   1:  PR[GP1:91,1] = PR[GP1:90,1] + 46.308;
   1:  PR[GP1:91,2] = PR[GP1:90,2] + 32.675;
   1:L PR[91] 10mm/sec CNT100;
   1:  PR[GP1:91,1] = PR[GP1:90,1] + 44.442;
   1:  PR[GP1:91,2] = PR[GP1:90,2] + 33.490;
   1:L PR[91] 10mm/sec CNT100;
   1:  PR[GP1:91,1] = PR[GP1:90,1] + 37.684;
   1:  PR[GP1:91,2] = PR[GP1:90,2] + 35.956;
   1:L PR[91] 10mm/sec CNT100;
   1:  PR[GP1:91,1] = PR[GP1:90,1] + 31.286;
   1:  PR[GP1:91,2] = PR[GP1:90,2] + 36.863;
   1:L PR[91] 10mm/sec CNT100;
   1:  PR[GP1:91,1] = PR[GP1:90,1] + 28.029;
   1:  PR[GP1:91,2] = PR[GP1:90,2] + 37.166;
   1:L PR[91] 10mm/sec CNT100;
   1:  PR[GP1:91,1] = PR[GP1:90,1] + 21.830;
   1:  PR[GP1:91,2] = PR[GP1:90,2] + 36.754;
   1:L PR[91] 10mm/sec CNT100;
   1:  PR[GP1:91,1] = PR[GP1:90,1] + 17.899;
   1:  PR[GP1:91,2] = PR[GP1:90,2] + 35.825;
   1:L PR[91] 10mm/sec CNT100;
   1:  PR[GP1:91,1] = PR[GP1:90,1] + 12.174;
   1:  PR[GP1:91,2] = PR[GP1:90,2] + 34.179;
   1:L PR[91] 10mm/sec CNT100;
   1:  PR[GP1:91,1] = PR[GP1:90,1] + 7.107;
   1:  PR[GP1:91,2] = PR[GP1:90,2] + 31.453;
   1:L PR[91] 10mm/sec CNT100;
   1:  PR[GP1:91,1] = PR[GP1:90,1] + -0.263;
   1:  PR[GP1:91,2] = PR[GP1:90,2] + 25.459;
   1:L PR[91] 10mm/sec CNT100;
   1:  PR[GP1:91,1] = PR[GP1:90,1] + -7.613;
   1:  PR[GP1:91,2] = PR[GP1:90,2] + 31.435;
   1:L PR[91] 10mm/sec CNT100;
   1:  PR[GP1:91,1] = PR[GP1:90,1] + -12.704;
   1:  PR[GP1:91,2] = PR[GP1:90,2] + 34.182;
   1:L PR[91] 10mm/sec CNT100;
   1:  PR[GP1:91,1] = PR[GP1:90,1] + -18.421;
   1:  PR[GP1:91,2] = PR[GP1:90,2] + 35.826;
   1:L PR[91] 10mm/sec CNT100;
   1:  PR[GP1:91,1] = PR[GP1:90,1] + -22.353;
   1:  PR[GP1:91,2] = PR[GP1:90,2] + 36.754;
   1:L PR[91] 10mm/sec CNT100;
   1:  PR[GP1:91,1] = PR[GP1:90,1] + -28.558;
   1:  PR[GP1:91,2] = PR[GP1:90,2] + 37.164;
   1:L PR[91] 10mm/sec CNT100;
   1:  PR[GP1:91,1] = PR[GP1:90,1] + -35.494;
   1:  PR[GP1:91,2] = PR[GP1:90,2] + 36.204;
   1:L PR[91] 10mm/sec CNT100;
   1:  PR[GP1:91,1] = PR[GP1:90,1] + -38.259;
   1:  PR[GP1:91,2] = PR[GP1:90,2] + 35.944;
   1:L PR[91] 10mm/sec CNT100;
   1:  PR[GP1:91,1] = PR[GP1:90,1] + -44.996;
   1:  PR[GP1:91,2] = PR[GP1:90,2] + 33.476;
   1:L PR[91] 10mm/sec CNT100;
   1:  PR[GP1:91,1] = PR[GP1:90,1] + -46.859;
   1:  PR[GP1:91,2] = PR[GP1:90,2] + 32.662;
   1:L PR[91] 10mm/sec CNT100;
   1:  PR[GP1:91,1] = PR[GP1:90,1] + -53.053;
   1:  PR[GP1:91,2] = PR[GP1:90,2] + 28.756;
   1:L PR[91] 10mm/sec CNT100;
   1:  PR[GP1:91,1] = PR[GP1:90,1] + -58.654;
   1:  PR[GP1:91,2] = PR[GP1:90,2] + 23.288;
   1:L PR[91] 10mm/sec CNT100;
   1:  PR[GP1:91,1] = PR[GP1:90,1] + -59.320;
   1:  PR[GP1:91,2] = PR[GP1:90,2] + 22.685;
   1:L PR[91] 10mm/sec CNT100;
   1:  PR[GP1:91,1] = PR[GP1:90,1] + -63.612;
   1:  PR[GP1:91,2] = PR[GP1:90,2] + 15.987;
   1:L PR[91] 10mm/sec CNT100;
   1:  PR[GP1:91,1] = PR[GP1:90,1] + -63.837;
   1:  PR[GP1:91,2] = PR[GP1:90,2] + 15.581;
   1:L PR[91] 10mm/sec CNT100;
   1:  PR[GP1:91,1] = PR[GP1:90,1] + -66.535;
   1:  PR[GP1:91,2] = PR[GP1:90,2] + 8.148;
   1:L PR[91] 10mm/sec CNT100;
   1:  PR[GP1:91,1] = PR[GP1:90,1] + -67.405;
   1:  PR[GP1:91,2] = PR[GP1:90,2] + 0.381;
   1:L PR[91] 10mm/sec CNT100;
   1:  PR[GP1:91,1] = PR[GP1:90,1] + -67.425;
   1:  PR[GP1:91,2] = PR[GP1:90,2] + 0.261;
   1:L PR[91] 10mm/sec CNT100;
   1:  PR[GP1:91,1] = PR[GP1:90,1] + -66.574;
   1:  PR[GP1:91,2] = PR[GP1:90,2] + -7.380;
   1:L PR[91] 10mm/sec CNT100;
   1:  PR[GP1:91,1] = PR[GP1:90,1] + -66.541;
   1:  PR[GP1:91,2] = PR[GP1:90,2] + -7.573;
   1:L PR[91] 10mm/sec CNT100;
   1:  PR[GP1:91,1] = PR[GP1:90,1] + -63.837;
   1:  PR[GP1:91,2] = PR[GP1:90,2] + -15.022;
   1:L PR[91] 10mm/sec CNT100;
   1:  PR[GP1:91,1] = PR[GP1:90,1] + -63.613;
   1:  PR[GP1:91,2] = PR[GP1:90,2] + -15.427;
   1:L PR[91] 10mm/sec CNT100;
   1:  PR[GP1:91,1] = PR[GP1:90,1] + -59.316;
   1:  PR[GP1:91,2] = PR[GP1:90,2] + -22.134;
   1:L PR[91] 10mm/sec CNT100;
   1:  PR[GP1:91,1] = PR[GP1:90,1] + -54.083;
   1:  PR[GP1:91,2] = PR[GP1:90,2] + -27.269;
   1:L PR[91] 10mm/sec CNT100;
   1:  PR[GP1:91,1] = PR[GP1:90,1] + -53.071;
   1:  PR[GP1:91,2] = PR[GP1:90,2] + -28.187;
   1:L PR[91] 10mm/sec CNT100;
   1:  PR[GP1:91,1] = PR[GP1:90,1] + -46.869;
   1:  PR[GP1:91,2] = PR[GP1:90,2] + -32.097;
   1:L PR[91] 10mm/sec CNT100;
   1:  PR[GP1:91,1] = PR[GP1:90,1] + -45.014;
   1:  PR[GP1:91,2] = PR[GP1:90,2] + -32.914;
   1:L PR[91] 10mm/sec CNT100;
   1:  PR[GP1:91,1] = PR[GP1:90,1] + -38.269;
   1:  PR[GP1:91,2] = PR[GP1:90,2] + -35.385;
   1:L PR[91] 10mm/sec CNT100;
   1:  PR[GP1:91,1] = PR[GP1:90,1] + -31.854;
   1:  PR[GP1:91,2] = PR[GP1:90,2] + -36.297;
   1:L PR[91] 10mm/sec CNT100;
   1:  PR[GP1:91,1] = PR[GP1:90,1] + -28.608;
   1:  PR[GP1:91,2] = PR[GP1:90,2] + -36.609;
   1:L PR[91] 10mm/sec CNT100;
   1:  PR[GP1:91,1] = PR[GP1:90,1] + -22.393;
   1:  PR[GP1:91,2] = PR[GP1:90,2] + -36.199;
   1:L PR[91] 10mm/sec CNT100;
   1:  PR[GP1:91,1] = PR[GP1:90,1] + -18.527;
   1:  PR[GP1:91,2] = PR[GP1:90,2] + -35.314;
   1:L PR[91] 10mm/sec CNT100;
   1:  PR[GP1:91,1] = PR[GP1:90,1] + -12.795;
   1:  PR[GP1:91,2] = PR[GP1:90,2] + -33.668;
   1:L PR[91] 10mm/sec CNT100;
   1:  PR[GP1:91,1] = PR[GP1:90,1] + -9.255;
   1:  PR[GP1:91,2] = PR[GP1:90,2] + -31.594;
   1:L PR[91] 10mm/sec CNT100;
   1:  PR[GP1:91,1] = PR[GP1:90,1] + -5.767;
   1:  PR[GP1:91,2] = PR[GP1:90,2] + -29.695;
   1:L PR[91] 10mm/sec CNT100;
   1:  PR[GP1:91,1] = PR[GP1:90,1] + -0.261;
   1:  PR[GP1:91,2] = PR[GP1:90,2] + -24.944;
   1:L PR[91] 10mm/sec CNT100;
   1:  PR[GP1:91,1] = PR[GP1:90,1] + 5.008;
   1:  PR[GP1:91,2] = PR[GP1:90,2] + -29.777;
   1:  PR[GP1:91,3] = PR[GP1:90,3] + 55.815;
   1:L PR[91] 10mm/sec CNT100;
   1:  PR[GP1:91,1] = PR[GP1:90,1] + 8.311;
   1:  PR[GP1:91,2] = PR[GP1:90,2] + -31.570;
   1:L PR[91] 10mm/sec CNT100;
   1:  PR[GP1:91,1] = PR[GP1:90,1] + 12.009;
   1:  PR[GP1:91,2] = PR[GP1:90,2] + -33.735;
   1:L PR[91] 10mm/sec CNT100;
   1:  PR[GP1:91,1] = PR[GP1:90,1] + 17.627;
   1:  PR[GP1:91,2] = PR[GP1:90,2] + -35.348;
   1:L PR[91] 10mm/sec CNT100;
   1:  PR[GP1:91,1] = PR[GP1:90,1] + 21.692;
   1:  PR[GP1:91,2] = PR[GP1:90,2] + -36.278;
   1:L PR[91] 10mm/sec CNT100;
   1:  PR[GP1:91,1] = PR[GP1:90,1] + 27.752;
   1:  PR[GP1:91,2] = PR[GP1:90,2] + -36.681;
   1:L PR[91] 10mm/sec CNT100;
   1:  PR[GP1:91,1] = PR[GP1:90,1] + 34.524;
   1:  PR[GP1:91,2] = PR[GP1:90,2] + -35.746;
   1:L PR[91] 10mm/sec CNT100;
   1:  PR[GP1:91,1] = PR[GP1:90,1] + 37.502;
   1:  PR[GP1:91,2] = PR[GP1:90,2] + -35.457;
   1:L PR[91] 10mm/sec CNT100;
   1:  PR[GP1:91,1] = PR[GP1:90,1] + 44.116;
   1:  PR[GP1:91,2] = PR[GP1:90,2] + -33.043;
   1:L PR[91] 10mm/sec CNT100;
   1:  PR[GP1:91,1] = PR[GP1:90,1] + 46.173;
   1:  PR[GP1:91,2] = PR[GP1:90,2] + -32.138;
   1:L PR[91] 10mm/sec CNT100;
   1:  PR[GP1:91,1] = PR[GP1:90,1] + 52.217;
   1:  PR[GP1:91,2] = PR[GP1:90,2] + -28.346;
   1:L PR[91] 10mm/sec CNT100;
   1:  PR[GP1:91,1] = PR[GP1:90,1] + 57.705;
   1:  PR[GP1:91,2] = PR[GP1:90,2] + -22.996;
   1:L PR[91] 10mm/sec CNT100;
   1:  PR[GP1:91,1] = PR[GP1:90,1] + 58.542;
   1:  PR[GP1:91,2] = PR[GP1:90,2] + -22.236;
   1:L PR[91] 10mm/sec CNT100;
   1:  PR[GP1:91,1] = PR[GP1:90,1] + 62.804;
   1:  PR[GP1:91,2] = PR[GP1:90,2] + -15.625;
   1:L PR[91] 10mm/sec CNT100;
   1:  PR[GP1:91,1] = PR[GP1:90,1] + 63.136;
   1:  PR[GP1:91,2] = PR[GP1:90,2] + -15.024;
   1:L PR[91] 10mm/sec CNT100;
   1:  PR[GP1:91,1] = PR[GP1:90,1] + 65.777;
   1:  PR[GP1:91,2] = PR[GP1:90,2] + -7.843;
   1:L PR[91] 10mm/sec CNT100;
   1:  PR[GP1:91,1] = PR[GP1:90,1] + 66.664;
   1:  PR[GP1:91,2] = PR[GP1:90,2] + -0.043;
   1:L PR[91] 10mm/sec CNT100;
   1:  PR[GP1:91,1] = PR[GP1:90,1] + 66.722;
   1:  PR[GP1:91,2] = PR[GP1:90,2] + 0.296;
   1:L PR[91] 10mm/sec CNT100;
   1:  PR[GP1:91,1] = PR[GP1:90,1] + 65.854;
   1:  PR[GP1:91,2] = PR[GP1:90,2] + 7.972;
   1:L PR[91] 10mm/sec CNT100;
   1:  PR[GP1:91,1] = PR[GP1:90,1] + 65.783;
   1:  PR[GP1:91,2] = PR[GP1:90,2] + 8.386;
   1:L PR[91] 10mm/sec CNT100;
   1:  PR[GP1:91,1] = PR[GP1:90,1] + 63.136;
   1:  PR[GP1:91,2] = PR[GP1:90,2] + 15.583;
   1:L PR[91] 10mm/sec CNT100;
   1:  PR[GP1:91,1] = PR[GP1:90,1] + 62.802;
   1:  PR[GP1:91,2] = PR[GP1:90,2] + 16.185;
   1:L PR[91] 10mm/sec CNT100;
   1:  PR[GP1:91,1] = PR[GP1:90,1] + 58.532;
   1:  PR[GP1:91,2] = PR[GP1:90,2] + 22.807;
   1:L PR[91] 10mm/sec CNT100;
   1:  PR[GP1:91,1] = PR[GP1:90,1] + 53.397;
   1:  PR[GP1:91,2] = PR[GP1:90,2] + 27.836;
   1:L PR[91] 10mm/sec CNT100;
   1:  PR[GP1:91,1] = PR[GP1:90,1] + 52.217;
   1:  PR[GP1:91,2] = PR[GP1:90,2] + 28.904;
   1:L PR[91] 10mm/sec CNT100;
   1:  PR[GP1:91,1] = PR[GP1:90,1] + 46.161;
   1:  PR[GP1:91,2] = PR[GP1:90,2] + 32.704;
   1:L PR[91] 10mm/sec CNT100;
   1:  PR[GP1:91,1] = PR[GP1:90,1] + 44.096;
   1:  PR[GP1:91,2] = PR[GP1:90,2] + 33.606;
   1:L PR[91] 10mm/sec CNT100;
   1:  PR[GP1:91,1] = PR[GP1:90,1] + 37.465;
   1:  PR[GP1:91,2] = PR[GP1:90,2] + 36.026;
   1:L PR[91] 10mm/sec CNT100;
   1:  PR[GP1:91,1] = PR[GP1:90,1] + 31.187;
   1:  PR[GP1:91,2] = PR[GP1:90,2] + 36.916;
   1:L PR[91] 10mm/sec CNT100;
   1:  PR[GP1:91,1] = PR[GP1:90,1] + 27.726;
   1:  PR[GP1:91,2] = PR[GP1:90,2] + 37.237;
   1:L PR[91] 10mm/sec CNT100;
   1:  PR[GP1:91,1] = PR[GP1:90,1] + 21.651;
   1:  PR[GP1:91,2] = PR[GP1:90,2] + 36.834;
   1:L PR[91] 10mm/sec CNT100;
   1:  PR[GP1:91,1] = PR[GP1:90,1] + 17.518;
   1:  PR[GP1:91,2] = PR[GP1:90,2] + 35.858;
   1:L PR[91] 10mm/sec CNT100;
   1:  PR[GP1:91,1] = PR[GP1:90,1] + 11.916;
   1:  PR[GP1:91,2] = PR[GP1:90,2] + 34.247;
   1:L PR[91] 10mm/sec CNT100;
   1:  PR[GP1:91,1] = PR[GP1:90,1] + 6.934;
   1:  PR[GP1:91,2] = PR[GP1:90,2] + 31.567;
   1:L PR[91] 10mm/sec CNT100;
   1:  PR[GP1:91,1] = PR[GP1:90,1] + -0.263;
   1:  PR[GP1:91,2] = PR[GP1:90,2] + 25.714;
   1:L PR[91] 10mm/sec CNT100;
   1:  PR[GP1:91,1] = PR[GP1:90,1] + -7.441;
   1:  PR[GP1:91,2] = PR[GP1:90,2] + 31.550;
   1:L PR[91] 10mm/sec CNT100;
   1:  PR[GP1:91,1] = PR[GP1:90,1] + -12.446;
   1:  PR[GP1:91,2] = PR[GP1:90,2] + 34.250;
   1:L PR[91] 10mm/sec CNT100;
   1:  PR[GP1:91,1] = PR[GP1:90,1] + -18.041;
   1:  PR[GP1:91,2] = PR[GP1:90,2] + 35.858;
   1:L PR[91] 10mm/sec CNT100;
   1:  PR[GP1:91,1] = PR[GP1:90,1] + -22.175;
   1:  PR[GP1:91,2] = PR[GP1:90,2] + 36.834;
   1:L PR[91] 10mm/sec CNT100;
   1:  PR[GP1:91,1] = PR[GP1:90,1] + -28.255;
   1:  PR[GP1:91,2] = PR[GP1:90,2] + 37.235;
   1:L PR[91] 10mm/sec CNT100;
   1:  PR[GP1:91,1] = PR[GP1:90,1] + -35.055;
   1:  PR[GP1:91,2] = PR[GP1:90,2] + 36.294;
   1:L PR[91] 10mm/sec CNT100;
   1:  PR[GP1:91,1] = PR[GP1:90,1] + -38.040;
   1:  PR[GP1:91,2] = PR[GP1:90,2] + 36.014;
   1:L PR[91] 10mm/sec CNT100;
   1:  PR[GP1:91,1] = PR[GP1:90,1] + -44.649;
   1:  PR[GP1:91,2] = PR[GP1:90,2] + 33.593;
   1:L PR[91] 10mm/sec CNT100;
   1:  PR[GP1:91,1] = PR[GP1:90,1] + -46.712;
   1:  PR[GP1:91,2] = PR[GP1:90,2] + 32.691;
   1:L PR[91] 10mm/sec CNT100;
   1:  PR[GP1:91,1] = PR[GP1:90,1] + -52.795;
   1:  PR[GP1:91,2] = PR[GP1:90,2] + 28.856;
   1:L PR[91] 10mm/sec CNT100;
   1:  PR[GP1:91,1] = PR[GP1:90,1] + -58.297;
   1:  PR[GP1:91,2] = PR[GP1:90,2] + 23.485;
   1:L PR[91] 10mm/sec CNT100;
   1:  PR[GP1:91,1] = PR[GP1:90,1] + -59.132;
   1:  PR[GP1:91,2] = PR[GP1:90,2] + 22.729;
   1:L PR[91] 10mm/sec CNT100;
   1:  PR[GP1:91,1] = PR[GP1:90,1] + -63.349;
   1:  PR[GP1:91,2] = PR[GP1:90,2] + 16.146;
   1:L PR[91] 10mm/sec CNT100;
   1:  PR[GP1:91,1] = PR[GP1:90,1] + -63.682;
   1:  PR[GP1:91,2] = PR[GP1:90,2] + 15.545;
   1:L PR[91] 10mm/sec CNT100;
   1:  PR[GP1:91,1] = PR[GP1:90,1] + -66.334;
   1:  PR[GP1:91,2] = PR[GP1:90,2] + 8.238;
   1:L PR[91] 10mm/sec CNT100;
   1:  PR[GP1:91,1] = PR[GP1:90,1] + -67.190;
   1:  PR[GP1:91,2] = PR[GP1:90,2] + 0.601;
   1:L PR[91] 10mm/sec CNT100;
   1:  PR[GP1:91,1] = PR[GP1:90,1] + -67.248;
   1:  PR[GP1:91,2] = PR[GP1:90,2] + 0.261;
   1:L PR[91] 10mm/sec CNT100;
   1:  PR[GP1:91,1] = PR[GP1:90,1] + -66.411;
   1:  PR[GP1:91,2] = PR[GP1:90,2] + -7.252;
   1:L PR[91] 10mm/sec CNT100;
   1:  PR[GP1:91,1] = PR[GP1:90,1] + -66.341;
   1:  PR[GP1:91,2] = PR[GP1:90,2] + -7.662;
   1:L PR[91] 10mm/sec CNT100;
   1:  PR[GP1:91,1] = PR[GP1:90,1] + -63.683;
   1:  PR[GP1:91,2] = PR[GP1:90,2] + -14.986;
   1:L PR[91] 10mm/sec CNT100;
   1:  PR[GP1:91,1] = PR[GP1:90,1] + -63.351;
   1:  PR[GP1:91,2] = PR[GP1:90,2] + -15.586;
   1:L PR[91] 10mm/sec CNT100;
   1:  PR[GP1:91,1] = PR[GP1:90,1] + -59.128;
   1:  PR[GP1:91,2] = PR[GP1:90,2] + -22.177;
   1:L PR[91] 10mm/sec CNT100;
   1:  PR[GP1:91,1] = PR[GP1:90,1] + -53.985;
   1:  PR[GP1:91,2] = PR[GP1:90,2] + -27.223;
   1:L PR[91] 10mm/sec CNT100;
   1:  PR[GP1:91,1] = PR[GP1:90,1] + -52.814;
   1:  PR[GP1:91,2] = PR[GP1:90,2] + -28.286;
   1:L PR[91] 10mm/sec CNT100;
   1:  PR[GP1:91,1] = PR[GP1:90,1] + -46.724;
   1:  PR[GP1:91,2] = PR[GP1:90,2] + -32.126;
   1:L PR[91] 10mm/sec CNT100;
   1:  PR[GP1:91,1] = PR[GP1:90,1] + -44.669;
   1:  PR[GP1:91,2] = PR[GP1:90,2] + -33.030;
   1:L PR[91] 10mm/sec CNT100;
   1:  PR[GP1:91,1] = PR[GP1:90,1] + -38.050;
   1:  PR[GP1:91,2] = PR[GP1:90,2] + -35.454;
   1:L PR[91] 10mm/sec CNT100;
   1:  PR[GP1:91,1] = PR[GP1:90,1] + -31.756;
   1:  PR[GP1:91,2] = PR[GP1:90,2] + -36.350;
   1:L PR[91] 10mm/sec CNT100;
   1:  PR[GP1:91,1] = PR[GP1:90,1] + -28.308;
   1:  PR[GP1:91,2] = PR[GP1:90,2] + -36.681;
   1:L PR[91] 10mm/sec CNT100;
   1:  PR[GP1:91,1] = PR[GP1:90,1] + -22.217;
   1:  PR[GP1:91,2] = PR[GP1:90,2] + -36.279;
   1:L PR[91] 10mm/sec CNT100;
   1:  PR[GP1:91,1] = PR[GP1:90,1] + -18.151;
   1:  PR[GP1:91,2] = PR[GP1:90,2] + -35.349;
   1:L PR[91] 10mm/sec CNT100;
   1:  PR[GP1:91,1] = PR[GP1:90,1] + -12.541;
   1:  PR[GP1:91,2] = PR[GP1:90,2] + -33.737;
   1:L PR[91] 10mm/sec CNT100;
   1:  PR[GP1:91,1] = PR[GP1:90,1] + -8.845;
   1:  PR[GP1:91,2] = PR[GP1:90,2] + -31.572;
   1:L PR[91] 10mm/sec CNT100;
   1:  PR[GP1:91,1] = PR[GP1:90,1] + -5.523;
   1:  PR[GP1:91,2] = PR[GP1:90,2] + -29.764;
   1:L PR[91] 10mm/sec CNT100;
   1:  PR[GP1:91,1] = PR[GP1:90,1] + -0.262;
   1:  PR[GP1:91,2] = PR[GP1:90,2] + -25.224;
   1:L PR[91] 10mm/sec CNT100;
   1:  PR[GP1:91,1] = PR[GP1:90,1] + 4.763;
   1:  PR[GP1:91,2] = PR[GP1:90,2] + -29.846;
   1:  PR[GP1:91,3] = PR[GP1:90,3] + 56.425;
   1:L PR[91] 10mm/sec CNT100;
   1:  PR[GP1:91,1] = PR[GP1:90,1] + 7.900;
   1:  PR[GP1:91,2] = PR[GP1:90,2] + -31.548;
   1:L PR[91] 10mm/sec CNT100;
   1:  PR[GP1:91,1] = PR[GP1:90,1] + 11.754;
   1:  PR[GP1:91,2] = PR[GP1:90,2] + -33.804;
   1:L PR[91] 10mm/sec CNT100;
   1:  PR[GP1:91,1] = PR[GP1:90,1] + 17.252;
   1:  PR[GP1:91,2] = PR[GP1:90,2] + -35.383;
   1:L PR[91] 10mm/sec CNT100;
   1:  PR[GP1:91,1] = PR[GP1:90,1] + 21.516;
   1:  PR[GP1:91,2] = PR[GP1:90,2] + -36.359;
   1:L PR[91] 10mm/sec CNT100;
   1:  PR[GP1:91,1] = PR[GP1:90,1] + 27.452;
   1:  PR[GP1:91,2] = PR[GP1:90,2] + -36.753;
   1:L PR[91] 10mm/sec CNT100;
   1:  PR[GP1:91,1] = PR[GP1:90,1] + 34.088;
   1:  PR[GP1:91,2] = PR[GP1:90,2] + -35.837;
   1:L PR[91] 10mm/sec CNT100;
   1:  PR[GP1:91,1] = PR[GP1:90,1] + 37.284;
   1:  PR[GP1:91,2] = PR[GP1:90,2] + -35.526;
   1:L PR[91] 10mm/sec CNT100;
   1:  PR[GP1:91,1] = PR[GP1:90,1] + 43.772;
   1:  PR[GP1:91,2] = PR[GP1:90,2] + -33.159;
   1:L PR[91] 10mm/sec CNT100;
   1:  PR[GP1:91,1] = PR[GP1:90,1] + 46.028;
   1:  PR[GP1:91,2] = PR[GP1:90,2] + -32.166;
   1:L PR[91] 10mm/sec CNT100;
   1:  PR[GP1:91,1] = PR[GP1:90,1] + 51.961;
   1:  PR[GP1:91,2] = PR[GP1:90,2] + -28.444;
   1:L PR[91] 10mm/sec CNT100;
   1:  PR[GP1:91,1] = PR[GP1:90,1] + 57.350;
   1:  PR[GP1:91,2] = PR[GP1:90,2] + -23.191;
   1:L PR[91] 10mm/sec CNT100;
   1:  PR[GP1:91,1] = PR[GP1:90,1] + 58.355;
   1:  PR[GP1:91,2] = PR[GP1:90,2] + -22.277;
   1:L PR[91] 10mm/sec CNT100;
   1:  PR[GP1:91,1] = PR[GP1:90,1] + 62.542;
   1:  PR[GP1:91,2] = PR[GP1:90,2] + -15.782;
   1:L PR[91] 10mm/sec CNT100;
   1:  PR[GP1:91,1] = PR[GP1:90,1] + 62.982;
   1:  PR[GP1:91,2] = PR[GP1:90,2] + -14.987;
   1:L PR[91] 10mm/sec CNT100;
   1:  PR[GP1:91,1] = PR[GP1:90,1] + 65.578;
   1:  PR[GP1:91,2] = PR[GP1:90,2] + -7.930;
   1:L PR[91] 10mm/sec CNT100;
   1:  PR[GP1:91,1] = PR[GP1:90,1] + 66.449;
   1:  PR[GP1:91,2] = PR[GP1:90,2] + -0.262;
   1:L PR[91] 10mm/sec CNT100;
   1:  PR[GP1:91,1] = PR[GP1:90,1] + 66.544;
   1:  PR[GP1:91,2] = PR[GP1:90,2] + 0.296;
   1:L PR[91] 10mm/sec CNT100;
   1:  PR[GP1:91,1] = PR[GP1:90,1] + 65.691;
   1:  PR[GP1:91,2] = PR[GP1:90,2] + 7.842;
   1:L PR[91] 10mm/sec CNT100;
   1:  PR[GP1:91,1] = PR[GP1:90,1] + 65.583;
   1:  PR[GP1:91,2] = PR[GP1:90,2] + 8.473;
   1:L PR[91] 10mm/sec CNT100;
   1:  PR[GP1:91,1] = PR[GP1:90,1] + 62.982;
   1:  PR[GP1:91,2] = PR[GP1:90,2] + 15.547;
   1:L PR[91] 10mm/sec CNT100;
   1:  PR[GP1:91,1] = PR[GP1:90,1] + 62.540;
   1:  PR[GP1:91,2] = PR[GP1:90,2] + 16.344;
   1:L PR[91] 10mm/sec CNT100;
   1:  PR[GP1:91,1] = PR[GP1:90,1] + 58.345;
   1:  PR[GP1:91,2] = PR[GP1:90,2] + 22.849;
   1:L PR[91] 10mm/sec CNT100;
   1:  PR[GP1:91,1] = PR[GP1:90,1] + 53.299;
   1:  PR[GP1:91,2] = PR[GP1:90,2] + 27.791;
   1:L PR[91] 10mm/sec CNT100;
   1:  PR[GP1:91,1] = PR[GP1:90,1] + 51.960;
   1:  PR[GP1:91,2] = PR[GP1:90,2] + 29.002;
   1:L PR[91] 10mm/sec CNT100;
   1:  PR[GP1:91,1] = PR[GP1:90,1] + 46.015;
   1:  PR[GP1:91,2] = PR[GP1:90,2] + 32.733;
   1:L PR[91] 10mm/sec CNT100;
   1:  PR[GP1:91,1] = PR[GP1:90,1] + 43.750;
   1:  PR[GP1:91,2] = PR[GP1:90,2] + 33.722;
   1:L PR[91] 10mm/sec CNT100;
   1:  PR[GP1:91,1] = PR[GP1:90,1] + 37.246;
   1:  PR[GP1:91,2] = PR[GP1:90,2] + 36.096;
   1:L PR[91] 10mm/sec CNT100;
   1:  PR[GP1:91,1] = PR[GP1:90,1] + 31.087;
   1:  PR[GP1:91,2] = PR[GP1:90,2] + 36.969;
   1:L PR[91] 10mm/sec CNT100;
   1:  PR[GP1:91,1] = PR[GP1:90,1] + 27.424;
   1:  PR[GP1:91,2] = PR[GP1:90,2] + 37.309;
   1:L PR[91] 10mm/sec CNT100;
   1:  PR[GP1:91,1] = PR[GP1:90,1] + 21.472;
   1:  PR[GP1:91,2] = PR[GP1:90,2] + 36.914;
   1:L PR[91] 10mm/sec CNT100;
   1:  PR[GP1:91,1] = PR[GP1:90,1] + 17.137;
   1:  PR[GP1:91,2] = PR[GP1:90,2] + 35.890;
   1:L PR[91] 10mm/sec CNT100;
   1:  PR[GP1:91,1] = PR[GP1:90,1] + 11.658;
   1:  PR[GP1:91,2] = PR[GP1:90,2] + 34.315;
   1:L PR[91] 10mm/sec CNT100;
   1:  PR[GP1:91,1] = PR[GP1:90,1] + 6.761;
   1:  PR[GP1:91,2] = PR[GP1:90,2] + 31.681;
   1:L PR[91] 10mm/sec CNT100;
   1:  PR[GP1:91,1] = PR[GP1:90,1] + -0.263;
   1:  PR[GP1:91,2] = PR[GP1:90,2] + 25.968;
   1:L PR[91] 10mm/sec CNT100;
   1:  PR[GP1:91,1] = PR[GP1:90,1] + -7.268;
   1:  PR[GP1:91,2] = PR[GP1:90,2] + 31.664;
   1:L PR[91] 10mm/sec CNT100;
   1:  PR[GP1:91,1] = PR[GP1:90,1] + -12.187;
   1:  PR[GP1:91,2] = PR[GP1:90,2] + 34.317;
   1:L PR[91] 10mm/sec CNT100;
   1:  PR[GP1:91,1] = PR[GP1:90,1] + -17.660;
   1:  PR[GP1:91,2] = PR[GP1:90,2] + 35.891;
   1:L PR[91] 10mm/sec CNT100;
   1:  PR[GP1:91,1] = PR[GP1:90,1] + -21.996;
   1:  PR[GP1:91,2] = PR[GP1:90,2] + 36.914;
   1:L PR[91] 10mm/sec CNT100;
   1:  PR[GP1:91,1] = PR[GP1:90,1] + -27.953;
   1:  PR[GP1:91,2] = PR[GP1:90,2] + 37.307;
   1:L PR[91] 10mm/sec CNT100;
   1:  PR[GP1:91,1] = PR[GP1:90,1] + -34.616;
   1:  PR[GP1:91,2] = PR[GP1:90,2] + 36.385;
   1:L PR[91] 10mm/sec CNT100;
   1:  PR[GP1:91,1] = PR[GP1:90,1] + -37.820;
   1:  PR[GP1:91,2] = PR[GP1:90,2] + 36.084;
   1:L PR[91] 10mm/sec CNT100;
   1:  PR[GP1:91,1] = PR[GP1:90,1] + -44.303;
   1:  PR[GP1:91,2] = PR[GP1:90,2] + 33.710;
   1:L PR[91] 10mm/sec CNT100;
   1:  PR[GP1:91,1] = PR[GP1:90,1] + -46.565;
   1:  PR[GP1:91,2] = PR[GP1:90,2] + 32.720;
   1:L PR[91] 10mm/sec CNT100;
   1:  PR[GP1:91,1] = PR[GP1:90,1] + -52.537;
   1:  PR[GP1:91,2] = PR[GP1:90,2] + 28.955;
   1:L PR[91] 10mm/sec CNT100;
   1:  PR[GP1:91,1] = PR[GP1:90,1] + -57.939;
   1:  PR[GP1:91,2] = PR[GP1:90,2] + 23.682;
   1:L PR[91] 10mm/sec CNT100;
   1:  PR[GP1:91,1] = PR[GP1:90,1] + -58.943;
   1:  PR[GP1:91,2] = PR[GP1:90,2] + 22.773;
   1:L PR[91] 10mm/sec CNT100;
   1:  PR[GP1:91,1] = PR[GP1:90,1] + -63.087;
   1:  PR[GP1:91,2] = PR[GP1:90,2] + 16.305;
   1:L PR[91] 10mm/sec CNT100;
   1:  PR[GP1:91,1] = PR[GP1:90,1] + -63.528;
   1:  PR[GP1:91,2] = PR[GP1:90,2] + 15.509;
   1:L PR[91] 10mm/sec CNT100;
   1:  PR[GP1:91,1] = PR[GP1:90,1] + -66.134;
   1:  PR[GP1:91,2] = PR[GP1:90,2] + 8.327;
   1:L PR[91] 10mm/sec CNT100;
   1:  PR[GP1:91,1] = PR[GP1:90,1] + -66.975;
   1:  PR[GP1:91,2] = PR[GP1:90,2] + 0.821;
   1:L PR[91] 10mm/sec CNT100;
   1:  PR[GP1:91,1] = PR[GP1:90,1] + -67.071;
   1:  PR[GP1:91,2] = PR[GP1:90,2] + 0.261;
   1:L PR[91] 10mm/sec CNT100;
   1:  PR[GP1:91,1] = PR[GP1:90,1] + -66.248;
   1:  PR[GP1:91,2] = PR[GP1:90,2] + -7.124;
   1:L PR[91] 10mm/sec CNT100;
   1:  PR[GP1:91,1] = PR[GP1:90,1] + -66.141;
   1:  PR[GP1:91,2] = PR[GP1:90,2] + -7.751;
   1:L PR[91] 10mm/sec CNT100;
   1:  PR[GP1:91,1] = PR[GP1:90,1] + -63.528;
   1:  PR[GP1:91,2] = PR[GP1:90,2] + -14.949;
   1:L PR[91] 10mm/sec CNT100;
   1:  PR[GP1:91,1] = PR[GP1:90,1] + -63.089;
   1:  PR[GP1:91,2] = PR[GP1:90,2] + -15.744;
   1:L PR[91] 10mm/sec CNT100;
   1:  PR[GP1:91,1] = PR[GP1:90,1] + -58.940;
   1:  PR[GP1:91,2] = PR[GP1:90,2] + -22.220;
   1:L PR[91] 10mm/sec CNT100;
   1:  PR[GP1:91,1] = PR[GP1:90,1] + -53.887;
   1:  PR[GP1:91,2] = PR[GP1:90,2] + -27.177;
   1:L PR[91] 10mm/sec CNT100;
   1:  PR[GP1:91,1] = PR[GP1:90,1] + -52.557;
   1:  PR[GP1:91,2] = PR[GP1:90,2] + -28.384;
   1:L PR[91] 10mm/sec CNT100;
   1:  PR[GP1:91,1] = PR[GP1:90,1] + -46.578;
   1:  PR[GP1:91,2] = PR[GP1:90,2] + -32.154;
   1:L PR[91] 10mm/sec CNT100;
   1:  PR[GP1:91,1] = PR[GP1:90,1] + -44.324;
   1:  PR[GP1:91,2] = PR[GP1:90,2] + -33.146;
   1:L PR[91] 10mm/sec CNT100;
   1:  PR[GP1:91,1] = PR[GP1:90,1] + -37.832;
   1:  PR[GP1:91,2] = PR[GP1:90,2] + -35.524;
   1:L PR[91] 10mm/sec CNT100;
   1:  PR[GP1:91,1] = PR[GP1:90,1] + -31.658;
   1:  PR[GP1:91,2] = PR[GP1:90,2] + -36.403;
   1:L PR[91] 10mm/sec CNT100;
   1:  PR[GP1:91,1] = PR[GP1:90,1] + -28.007;
   1:  PR[GP1:91,2] = PR[GP1:90,2] + -36.753;
   1:L PR[91] 10mm/sec CNT100;
   1:  PR[GP1:91,1] = PR[GP1:90,1] + -22.040;
   1:  PR[GP1:91,2] = PR[GP1:90,2] + -36.359;
   1:L PR[91] 10mm/sec CNT100;
   1:  PR[GP1:91,1] = PR[GP1:90,1] + -17.776;
   1:  PR[GP1:91,2] = PR[GP1:90,2] + -35.383;
   1:L PR[91] 10mm/sec CNT100;
   1:  PR[GP1:91,1] = PR[GP1:90,1] + -12.286;
   1:  PR[GP1:91,2] = PR[GP1:90,2] + -33.807;
   1:L PR[91] 10mm/sec CNT100;
   1:  PR[GP1:91,1] = PR[GP1:90,1] + -8.434;
   1:  PR[GP1:91,2] = PR[GP1:90,2] + -31.550;
   1:L PR[91] 10mm/sec CNT100;
   1:  PR[GP1:91,1] = PR[GP1:90,1] + -5.280;
   1:  PR[GP1:91,2] = PR[GP1:90,2] + -29.833;
   1:L PR[91] 10mm/sec CNT100;
   1:  PR[GP1:91,1] = PR[GP1:90,1] + -0.262;
   1:  PR[GP1:91,2] = PR[GP1:90,2] + -25.503;
   1:L PR[91] 10mm/sec CNT100;
   1:  PR[GP1:91,1] = PR[GP1:90,1] + 4.519;
   1:  PR[GP1:91,2] = PR[GP1:90,2] + -29.914;
   1:  PR[GP1:91,3] = PR[GP1:90,3] + 57.035;
   1:L PR[91] 10mm/sec CNT100;
   1:  PR[GP1:91,1] = PR[GP1:90,1] + 7.489;
   1:  PR[GP1:91,2] = PR[GP1:90,2] + -31.526;
   1:L PR[91] 10mm/sec CNT100;
   1:  PR[GP1:91,1] = PR[GP1:90,1] + 11.500;
   1:  PR[GP1:91,2] = PR[GP1:90,2] + -33.874;
   1:L PR[91] 10mm/sec CNT100;
   1:  PR[GP1:91,1] = PR[GP1:90,1] + 16.876;
   1:  PR[GP1:91,2] = PR[GP1:90,2] + -35.418;
   1:L PR[91] 10mm/sec CNT100;
   1:  PR[GP1:91,1] = PR[GP1:90,1] + 21.339;
   1:  PR[GP1:91,2] = PR[GP1:90,2] + -36.439;
   1:L PR[91] 10mm/sec CNT100;
   1:  PR[GP1:91,1] = PR[GP1:90,1] + 27.152;
   1:  PR[GP1:91,2] = PR[GP1:90,2] + -36.825;
   1:L PR[91] 10mm/sec CNT100;
   1:  PR[GP1:91,1] = PR[GP1:90,1] + 33.652;
   1:  PR[GP1:91,2] = PR[GP1:90,2] + -35.928;
   1:L PR[91] 10mm/sec CNT100;
   1:  PR[GP1:91,1] = PR[GP1:90,1] + 37.067;
   1:  PR[GP1:91,2] = PR[GP1:90,2] + -35.596;
   1:L PR[91] 10mm/sec CNT100;
   1:  PR[GP1:91,1] = PR[GP1:90,1] + 43.427;
   1:  PR[GP1:91,2] = PR[GP1:90,2] + -33.274;
   1:L PR[91] 10mm/sec CNT100;
   1:  PR[GP1:91,1] = PR[GP1:90,1] + 45.882;
   1:  PR[GP1:91,2] = PR[GP1:90,2] + -32.195;
   1:L PR[91] 10mm/sec CNT100;
   1:  PR[GP1:91,1] = PR[GP1:90,1] + 51.706;
   1:  PR[GP1:91,2] = PR[GP1:90,2] + -28.541;
   1:L PR[91] 10mm/sec CNT100;
   1:  PR[GP1:91,1] = PR[GP1:90,1] + 56.995;
   1:  PR[GP1:91,2] = PR[GP1:90,2] + -23.385;
   1:L PR[91] 10mm/sec CNT100;
   1:  PR[GP1:91,1] = PR[GP1:90,1] + 58.168;
   1:  PR[GP1:91,2] = PR[GP1:90,2] + -22.319;
   1:L PR[91] 10mm/sec CNT100;
   1:  PR[GP1:91,1] = PR[GP1:90,1] + 62.280;
   1:  PR[GP1:91,2] = PR[GP1:90,2] + -15.940;
   1:L PR[91] 10mm/sec CNT100;
   1:  PR[GP1:91,1] = PR[GP1:90,1] + 62.828;
   1:  PR[GP1:91,2] = PR[GP1:90,2] + -14.950;
   1:L PR[91] 10mm/sec CNT100;
   1:  PR[GP1:91,1] = PR[GP1:90,1] + 65.378;
   1:  PR[GP1:91,2] = PR[GP1:90,2] + -8.017;
   1:L PR[91] 10mm/sec CNT100;
   1:  PR[GP1:91,1] = PR[GP1:90,1] + 66.234;
   1:  PR[GP1:91,2] = PR[GP1:90,2] + -0.482;
   1:L PR[91] 10mm/sec CNT100;
   1:  PR[GP1:91,1] = PR[GP1:90,1] + 66.367;
   1:  PR[GP1:91,2] = PR[GP1:90,2] + 0.296;
   1:L PR[91] 10mm/sec CNT100;
   1:  PR[GP1:91,1] = PR[GP1:90,1] + 65.529;
   1:  PR[GP1:91,2] = PR[GP1:90,2] + 7.711;
   1:L PR[91] 10mm/sec CNT100;
   1:  PR[GP1:91,1] = PR[GP1:90,1] + 65.383;
   1:  PR[GP1:91,2] = PR[GP1:90,2] + 8.560;
   1:L PR[91] 10mm/sec CNT100;
   1:  PR[GP1:91,1] = PR[GP1:90,1] + 62.827;
   1:  PR[GP1:91,2] = PR[GP1:90,2] + 15.510;
   1:L PR[91] 10mm/sec CNT100;
   1:  PR[GP1:91,1] = PR[GP1:90,1] + 62.277;
   1:  PR[GP1:91,2] = PR[GP1:90,2] + 16.502;
   1:L PR[91] 10mm/sec CNT100;
   1:  PR[GP1:91,1] = PR[GP1:90,1] + 58.158;
   1:  PR[GP1:91,2] = PR[GP1:90,2] + 22.892;
   1:L PR[91] 10mm/sec CNT100;
   1:  PR[GP1:91,1] = PR[GP1:90,1] + 53.202;
   1:  PR[GP1:91,2] = PR[GP1:90,2] + 27.745;
   1:L PR[91] 10mm/sec CNT100;
   1:  PR[GP1:91,1] = PR[GP1:90,1] + 51.703;
   1:  PR[GP1:91,2] = PR[GP1:90,2] + 29.101;
   1:L PR[91] 10mm/sec CNT100;
   1:  PR[GP1:91,1] = PR[GP1:90,1] + 45.869;
   1:  PR[GP1:91,2] = PR[GP1:90,2] + 32.762;
   1:L PR[91] 10mm/sec CNT100;
   1:  PR[GP1:91,1] = PR[GP1:90,1] + 43.404;
   1:  PR[GP1:91,2] = PR[GP1:90,2] + 33.838;
   1:L PR[91] 10mm/sec CNT100;
   1:  PR[GP1:91,1] = PR[GP1:90,1] + 37.026;
   1:  PR[GP1:91,2] = PR[GP1:90,2] + 36.166;
   1:L PR[91] 10mm/sec CNT100;
   1:  PR[GP1:91,1] = PR[GP1:90,1] + 30.988;
   1:  PR[GP1:91,2] = PR[GP1:90,2] + 37.022;
   1:L PR[91] 10mm/sec CNT100;
   1:  PR[GP1:91,1] = PR[GP1:90,1] + 27.122;
   1:  PR[GP1:91,2] = PR[GP1:90,2] + 37.381;
   1:L PR[91] 10mm/sec CNT100;
   1:  PR[GP1:91,1] = PR[GP1:90,1] + 21.293;
   1:  PR[GP1:91,2] = PR[GP1:90,2] + 36.994;
   1:L PR[91] 10mm/sec CNT100;
   1:  PR[GP1:91,1] = PR[GP1:90,1] + 16.757;
   1:  PR[GP1:91,2] = PR[GP1:90,2] + 35.923;
   1:L PR[91] 10mm/sec CNT100;
   1:  PR[GP1:91,1] = PR[GP1:90,1] + 11.399;
   1:  PR[GP1:91,2] = PR[GP1:90,2] + 34.382;
   1:L PR[91] 10mm/sec CNT100;
   1:  PR[GP1:91,1] = PR[GP1:90,1] + 6.588;
   1:  PR[GP1:91,2] = PR[GP1:90,2] + 31.795;
   1:L PR[91] 10mm/sec CNT100;
   1:  PR[GP1:91,1] = PR[GP1:90,1] + -0.263;
   1:  PR[GP1:91,2] = PR[GP1:90,2] + 26.223;
   1:L PR[91] 10mm/sec CNT100;
   1:  PR[GP1:91,1] = PR[GP1:90,1] + -7.096;
   1:  PR[GP1:91,2] = PR[GP1:90,2] + 31.779;
   1:L PR[91] 10mm/sec CNT100;
   1:  PR[GP1:91,1] = PR[GP1:90,1] + -11.929;
   1:  PR[GP1:91,2] = PR[GP1:90,2] + 34.385;
   1:L PR[91] 10mm/sec CNT100;
   1:  PR[GP1:91,1] = PR[GP1:90,1] + -17.279;
   1:  PR[GP1:91,2] = PR[GP1:90,2] + 35.923;
   1:L PR[91] 10mm/sec CNT100;
   1:  PR[GP1:91,1] = PR[GP1:90,1] + -21.817;
   1:  PR[GP1:91,2] = PR[GP1:90,2] + 36.994;
   1:L PR[91] 10mm/sec CNT100;
   1:  PR[GP1:91,1] = PR[GP1:90,1] + -27.650;
   1:  PR[GP1:91,2] = PR[GP1:90,2] + 37.379;
   1:L PR[91] 10mm/sec CNT100;
   1:  PR[GP1:91,1] = PR[GP1:90,1] + -34.176;
   1:  PR[GP1:91,2] = PR[GP1:90,2] + 36.476;
   1:L PR[91] 10mm/sec CNT100;
   1:  PR[GP1:91,1] = PR[GP1:90,1] + -37.600;
   1:  PR[GP1:91,2] = PR[GP1:90,2] + 36.154;
   1:L PR[91] 10mm/sec CNT100;
   1:  PR[GP1:91,1] = PR[GP1:90,1] + -43.956;
   1:  PR[GP1:91,2] = PR[GP1:90,2] + 33.826;
   1:L PR[91] 10mm/sec CNT100;
   1:  PR[GP1:91,1] = PR[GP1:90,1] + -46.419;
   1:  PR[GP1:91,2] = PR[GP1:90,2] + 32.750;
   1:L PR[91] 10mm/sec CNT100;
   1:  PR[GP1:91,1] = PR[GP1:90,1] + -52.279;
   1:  PR[GP1:91,2] = PR[GP1:90,2] + 29.054;
   1:L PR[91] 10mm/sec CNT100;
   1:  PR[GP1:91,1] = PR[GP1:90,1] + -57.581;
   1:  PR[GP1:91,2] = PR[GP1:90,2] + 23.878;
   1:L PR[91] 10mm/sec CNT100;
   1:  PR[GP1:91,1] = PR[GP1:90,1] + -58.755;
   1:  PR[GP1:91,2] = PR[GP1:90,2] + 22.816;
   1:L PR[91] 10mm/sec CNT100;
   1:  PR[GP1:91,1] = PR[GP1:90,1] + -62.824;
   1:  PR[GP1:91,2] = PR[GP1:90,2] + 16.465;
   1:L PR[91] 10mm/sec CNT100;
   1:  PR[GP1:91,1] = PR[GP1:90,1] + -63.373;
   1:  PR[GP1:91,2] = PR[GP1:90,2] + 15.473;
   1:L PR[91] 10mm/sec CNT100;
   1:  PR[GP1:91,1] = PR[GP1:90,1] + -65.934;
   1:  PR[GP1:91,2] = PR[GP1:90,2] + 8.417;
   1:L PR[91] 10mm/sec CNT100;
   1:  PR[GP1:91,1] = PR[GP1:90,1] + -66.760;
   1:  PR[GP1:91,2] = PR[GP1:90,2] + 1.041;
   1:L PR[91] 10mm/sec CNT100;
   1:  PR[GP1:91,1] = PR[GP1:90,1] + -66.894;
   1:  PR[GP1:91,2] = PR[GP1:90,2] + 0.261;
   1:L PR[91] 10mm/sec CNT100;
   1:  PR[GP1:91,1] = PR[GP1:90,1] + -66.085;
   1:  PR[GP1:91,2] = PR[GP1:90,2] + -6.996;
   1:L PR[91] 10mm/sec CNT100;
   1:  PR[GP1:91,1] = PR[GP1:90,1] + -65.941;
   1:  PR[GP1:91,2] = PR[GP1:90,2] + -7.841;
   1:L PR[91] 10mm/sec CNT100;
   1:  PR[GP1:91,1] = PR[GP1:90,1] + -63.374;
   1:  PR[GP1:91,2] = PR[GP1:90,2] + -14.913;
   1:L PR[91] 10mm/sec CNT100;
   1:  PR[GP1:91,1] = PR[GP1:90,1] + -62.827;
   1:  PR[GP1:91,2] = PR[GP1:90,2] + -15.902;
   1:L PR[91] 10mm/sec CNT100;
   1:  PR[GP1:91,1] = PR[GP1:90,1] + -58.752;
   1:  PR[GP1:91,2] = PR[GP1:90,2] + -22.263;
   1:L PR[91] 10mm/sec CNT100;
   1:  PR[GP1:91,1] = PR[GP1:90,1] + -53.789;
   1:  PR[GP1:91,2] = PR[GP1:90,2] + -27.132;
   1:L PR[91] 10mm/sec CNT100;
   1:  PR[GP1:91,1] = PR[GP1:90,1] + -52.300;
   1:  PR[GP1:91,2] = PR[GP1:90,2] + -28.483;
   1:L PR[91] 10mm/sec CNT100;
   1:  PR[GP1:91,1] = PR[GP1:90,1] + -46.432;
   1:  PR[GP1:91,2] = PR[GP1:90,2] + -32.183;
   1:L PR[91] 10mm/sec CNT100;
   1:  PR[GP1:91,1] = PR[GP1:90,1] + -43.980;
   1:  PR[GP1:91,2] = PR[GP1:90,2] + -33.262;
   1:L PR[91] 10mm/sec CNT100;
   1:  PR[GP1:91,1] = PR[GP1:90,1] + -37.614;
   1:  PR[GP1:91,2] = PR[GP1:90,2] + -35.594;
   1:L PR[91] 10mm/sec CNT100;
   1:  PR[GP1:91,1] = PR[GP1:90,1] + -31.560;
   1:  PR[GP1:91,2] = PR[GP1:90,2] + -36.455;
   1:L PR[91] 10mm/sec CNT100;
   1:  PR[GP1:91,1] = PR[GP1:90,1] + -27.707;
   1:  PR[GP1:91,2] = PR[GP1:90,2] + -36.825;
   1:L PR[91] 10mm/sec CNT100;
   1:  PR[GP1:91,1] = PR[GP1:90,1] + -21.863;
   1:  PR[GP1:91,2] = PR[GP1:90,2] + -36.439;
   1:L PR[91] 10mm/sec CNT100;
   1:  PR[GP1:91,1] = PR[GP1:90,1] + -17.401;
   1:  PR[GP1:91,2] = PR[GP1:90,2] + -35.418;
   1:L PR[91] 10mm/sec CNT100;
   1:  PR[GP1:91,1] = PR[GP1:90,1] + -12.031;
   1:  PR[GP1:91,2] = PR[GP1:90,2] + -33.876;
   1:L PR[91] 10mm/sec CNT100;
   1:  PR[GP1:91,1] = PR[GP1:90,1] + -8.024;
   1:  PR[GP1:91,2] = PR[GP1:90,2] + -31.528;
   1:L PR[91] 10mm/sec CNT100;
   1:  PR[GP1:91,1] = PR[GP1:90,1] + -5.036;
   1:  PR[GP1:91,2] = PR[GP1:90,2] + -29.902;
   1:L PR[91] 10mm/sec CNT100;
   1:  PR[GP1:91,1] = PR[GP1:90,1] + -0.262;
   1:  PR[GP1:91,2] = PR[GP1:90,2] + -25.782;
   1:L PR[91] 10mm/sec CNT100;
   1:  PR[GP1:91,1] = PR[GP1:90,1] + 4.274;
   1:  PR[GP1:91,2] = PR[GP1:90,2] + -29.982;
   1:  PR[GP1:91,3] = PR[GP1:90,3] + 57.645;
   1:L PR[91] 10mm/sec CNT100;
   1:  PR[GP1:91,1] = PR[GP1:90,1] + 7.079;
   1:  PR[GP1:91,2] = PR[GP1:90,2] + -31.505;
   1:L PR[91] 10mm/sec CNT100;
   1:  PR[GP1:91,1] = PR[GP1:90,1] + 11.245;
   1:  PR[GP1:91,2] = PR[GP1:90,2] + -33.943;
   1:L PR[91] 10mm/sec CNT100;
   1:  PR[GP1:91,1] = PR[GP1:90,1] + 16.501;
   1:  PR[GP1:91,2] = PR[GP1:90,2] + -35.453;
   1:L PR[91] 10mm/sec CNT100;
   1:  PR[GP1:91,1] = PR[GP1:90,1] + 21.162;
   1:  PR[GP1:91,2] = PR[GP1:90,2] + -36.519;
   1:L PR[91] 10mm/sec CNT100;
   1:  PR[GP1:91,1] = PR[GP1:90,1] + 26.853;
   1:  PR[GP1:91,2] = PR[GP1:90,2] + -36.897;
   1:L PR[91] 10mm/sec CNT100;
   1:  PR[GP1:91,1] = PR[GP1:90,1] + 33.216;
   1:  PR[GP1:91,2] = PR[GP1:90,2] + -36.019;
   1:L PR[91] 10mm/sec CNT100;
   1:  PR[GP1:91,1] = PR[GP1:90,1] + 36.849;
   1:  PR[GP1:91,2] = PR[GP1:90,2] + -35.666;
   1:L PR[91] 10mm/sec CNT100;
   1:  PR[GP1:91,1] = PR[GP1:90,1] + 43.083;
   1:  PR[GP1:91,2] = PR[GP1:90,2] + -33.390;
   1:L PR[91] 10mm/sec CNT100;
   1:  PR[GP1:91,1] = PR[GP1:90,1] + 45.737;
   1:  PR[GP1:91,2] = PR[GP1:90,2] + -32.223;
   1:L PR[91] 10mm/sec CNT100;
   1:  PR[GP1:91,1] = PR[GP1:90,1] + 51.450;
   1:  PR[GP1:91,2] = PR[GP1:90,2] + -28.639;
   1:L PR[91] 10mm/sec CNT100;
   1:  PR[GP1:91,1] = PR[GP1:90,1] + 56.640;
   1:  PR[GP1:91,2] = PR[GP1:90,2] + -23.580;
   1:L PR[91] 10mm/sec CNT100;
   1:  PR[GP1:91,1] = PR[GP1:90,1] + 57.981;
   1:  PR[GP1:91,2] = PR[GP1:90,2] + -22.360;
   1:L PR[91] 10mm/sec CNT100;
   1:  PR[GP1:91,1] = PR[GP1:90,1] + 62.019;
   1:  PR[GP1:91,2] = PR[GP1:90,2] + -16.098;
   1:L PR[91] 10mm/sec CNT100;
   1:  PR[GP1:91,1] = PR[GP1:90,1] + 62.674;
   1:  PR[GP1:91,2] = PR[GP1:90,2] + -14.913;
   1:L PR[91] 10mm/sec CNT100;
   1:  PR[GP1:91,1] = PR[GP1:90,1] + 65.179;
   1:  PR[GP1:91,2] = PR[GP1:90,2] + -8.103;
   1:L PR[91] 10mm/sec CNT100;
   1:  PR[GP1:91,1] = PR[GP1:90,1] + 66.020;
   1:  PR[GP1:91,2] = PR[GP1:90,2] + -0.702;
   1:L PR[91] 10mm/sec CNT100;
   1:  PR[GP1:91,1] = PR[GP1:90,1] + 66.190;
   1:  PR[GP1:91,2] = PR[GP1:90,2] + 0.296;
   1:L PR[91] 10mm/sec CNT100;
   1:  PR[GP1:91,1] = PR[GP1:90,1] + 65.366;
   1:  PR[GP1:91,2] = PR[GP1:90,2] + 7.581;
   1:L PR[91] 10mm/sec CNT100;
   1:  PR[GP1:91,1] = PR[GP1:90,1] + 65.184;
   1:  PR[GP1:91,2] = PR[GP1:90,2] + 8.648;
   1:L PR[91] 10mm/sec CNT100;
   1:  PR[GP1:91,1] = PR[GP1:90,1] + 62.673;
   1:  PR[GP1:91,2] = PR[GP1:90,2] + 15.474;
   1:L PR[91] 10mm/sec CNT100;
   1:  PR[GP1:91,1] = PR[GP1:90,1] + 62.015;
   1:  PR[GP1:91,2] = PR[GP1:90,2] + 16.660;
   1:L PR[91] 10mm/sec CNT100;
   1:  PR[GP1:91,1] = PR[GP1:90,1] + 57.970;
   1:  PR[GP1:91,2] = PR[GP1:90,2] + 22.934;
   1:L PR[91] 10mm/sec CNT100;
   1:  PR[GP1:91,1] = PR[GP1:90,1] + 53.104;
   1:  PR[GP1:91,2] = PR[GP1:90,2] + 27.699;
   1:L PR[91] 10mm/sec CNT100;
   1:  PR[GP1:91,1] = PR[GP1:90,1] + 51.447;
   1:  PR[GP1:91,2] = PR[GP1:90,2] + 29.199;
   1:L PR[91] 10mm/sec CNT100;
   1:  PR[GP1:91,1] = PR[GP1:90,1] + 45.722;
   1:  PR[GP1:91,2] = PR[GP1:90,2] + 32.791;
   1:L PR[91] 10mm/sec CNT100;
   1:  PR[GP1:91,1] = PR[GP1:90,1] + 43.058;
   1:  PR[GP1:91,2] = PR[GP1:90,2] + 33.955;
   1:L PR[91] 10mm/sec CNT100;
   1:  PR[GP1:91,1] = PR[GP1:90,1] + 36.807;
   1:  PR[GP1:91,2] = PR[GP1:90,2] + 36.236;
   1:L PR[91] 10mm/sec CNT100;
   1:  PR[GP1:91,1] = PR[GP1:90,1] + 30.889;
   1:  PR[GP1:91,2] = PR[GP1:90,2] + 37.075;
   1:L PR[91] 10mm/sec CNT100;
   1:  PR[GP1:91,1] = PR[GP1:90,1] + 26.820;
   1:  PR[GP1:91,2] = PR[GP1:90,2] + 37.453;
   1:L PR[91] 10mm/sec CNT100;
   1:  PR[GP1:91,1] = PR[GP1:90,1] + 21.114;
   1:  PR[GP1:91,2] = PR[GP1:90,2] + 37.074;
   1:L PR[91] 10mm/sec CNT100;
   1:  PR[GP1:91,1] = PR[GP1:90,1] + 16.376;
   1:  PR[GP1:91,2] = PR[GP1:90,2] + 35.955;
   1:L PR[91] 10mm/sec CNT100;
   1:  PR[GP1:91,1] = PR[GP1:90,1] + 11.141;
   1:  PR[GP1:91,2] = PR[GP1:90,2] + 34.450;
   1:L PR[91] 10mm/sec CNT100;
   1:  PR[GP1:91,1] = PR[GP1:90,1] + 6.415;
   1:  PR[GP1:91,2] = PR[GP1:90,2] + 31.909;
   1:L PR[91] 10mm/sec CNT100;
   1:  PR[GP1:91,1] = PR[GP1:90,1] + -0.263;
   1:  PR[GP1:91,2] = PR[GP1:90,2] + 26.478;
   1:L PR[91] 10mm/sec CNT100;
   1:  PR[GP1:91,1] = PR[GP1:90,1] + -6.924;
   1:  PR[GP1:91,2] = PR[GP1:90,2] + 31.893;
   1:L PR[91] 10mm/sec CNT100;
   1:  PR[GP1:91,1] = PR[GP1:90,1] + -11.671;
   1:  PR[GP1:91,2] = PR[GP1:90,2] + 34.453;
   1:L PR[91] 10mm/sec CNT100;
   1:  PR[GP1:91,1] = PR[GP1:90,1] + -16.898;
   1:  PR[GP1:91,2] = PR[GP1:90,2] + 35.955;
   1:L PR[91] 10mm/sec CNT100;
   1:  PR[GP1:91,1] = PR[GP1:90,1] + -21.638;
   1:  PR[GP1:91,2] = PR[GP1:90,2] + 37.074;
   1:L PR[91] 10mm/sec CNT100;
   1:  PR[GP1:91,1] = PR[GP1:90,1] + -27.348;
   1:  PR[GP1:91,2] = PR[GP1:90,2] + 37.451;
   1:L PR[91] 10mm/sec CNT100;
   1:  PR[GP1:91,1] = PR[GP1:90,1] + -33.737;
   1:  PR[GP1:91,2] = PR[GP1:90,2] + 36.567;
   1:L PR[91] 10mm/sec CNT100;
   1:  PR[GP1:91,1] = PR[GP1:90,1] + -37.380;
   1:  PR[GP1:91,2] = PR[GP1:90,2] + 36.224;
   1:L PR[91] 10mm/sec CNT100;
   1:  PR[GP1:91,1] = PR[GP1:90,1] + -43.610;
   1:  PR[GP1:91,2] = PR[GP1:90,2] + 33.943;
   1:L PR[91] 10mm/sec CNT100;
   1:  PR[GP1:91,1] = PR[GP1:90,1] + -46.272;
   1:  PR[GP1:91,2] = PR[GP1:90,2] + 32.779;
   1:L PR[91] 10mm/sec CNT100;
   1:  PR[GP1:91,1] = PR[GP1:90,1] + -52.021;
   1:  PR[GP1:91,2] = PR[GP1:90,2] + 29.154;
   1:L PR[91] 10mm/sec CNT100;
   1:  PR[GP1:91,1] = PR[GP1:90,1] + -57.224;
   1:  PR[GP1:91,2] = PR[GP1:90,2] + 24.075;
   1:L PR[91] 10mm/sec CNT100;
   1:  PR[GP1:91,1] = PR[GP1:90,1] + -58.566;
   1:  PR[GP1:91,2] = PR[GP1:90,2] + 22.860;
   1:L PR[91] 10mm/sec CNT100;
   1:  PR[GP1:91,1] = PR[GP1:90,1] + -62.561;
   1:  PR[GP1:91,2] = PR[GP1:90,2] + 16.624;
   1:L PR[91] 10mm/sec CNT100;
   1:  PR[GP1:91,1] = PR[GP1:90,1] + -63.218;
   1:  PR[GP1:91,2] = PR[GP1:90,2] + 15.437;
   1:L PR[91] 10mm/sec CNT100;
   1:  PR[GP1:91,1] = PR[GP1:90,1] + -65.734;
   1:  PR[GP1:91,2] = PR[GP1:90,2] + 8.507;
   1:L PR[91] 10mm/sec CNT100;
   1:  PR[GP1:91,1] = PR[GP1:90,1] + -66.545;
   1:  PR[GP1:91,2] = PR[GP1:90,2] + 1.261;
   1:L PR[91] 10mm/sec CNT100;
   1:  PR[GP1:91,1] = PR[GP1:90,1] + -66.716;
   1:  PR[GP1:91,2] = PR[GP1:90,2] + 0.261;
   1:L PR[91] 10mm/sec CNT100;
   1:  PR[GP1:91,1] = PR[GP1:90,1] + -65.922;
   1:  PR[GP1:91,2] = PR[GP1:90,2] + -6.868;
   1:L PR[91] 10mm/sec CNT100;
   1:  PR[GP1:91,1] = PR[GP1:90,1] + -65.740;
   1:  PR[GP1:91,2] = PR[GP1:90,2] + -7.930;
   1:L PR[91] 10mm/sec CNT100;
   1:  PR[GP1:91,1] = PR[GP1:90,1] + -63.219;
   1:  PR[GP1:91,2] = PR[GP1:90,2] + -14.876;
   1:L PR[91] 10mm/sec CNT100;
   1:  PR[GP1:91,1] = PR[GP1:90,1] + -62.565;
   1:  PR[GP1:91,2] = PR[GP1:90,2] + -16.061;
   1:L PR[91] 10mm/sec CNT100;
   1:  PR[GP1:91,1] = PR[GP1:90,1] + -58.564;
   1:  PR[GP1:91,2] = PR[GP1:90,2] + -22.306;
   1:L PR[91] 10mm/sec CNT100;
   1:  PR[GP1:91,1] = PR[GP1:90,1] + -53.692;
   1:  PR[GP1:91,2] = PR[GP1:90,2] + -27.086;
   1:L PR[91] 10mm/sec CNT100;
   1:  PR[GP1:91,1] = PR[GP1:90,1] + -52.044;
   1:  PR[GP1:91,2] = PR[GP1:90,2] + -28.581;
   1:L PR[91] 10mm/sec CNT100;
   1:  PR[GP1:91,1] = PR[GP1:90,1] + -46.287;
   1:  PR[GP1:91,2] = PR[GP1:90,2] + -32.211;
   1:L PR[91] 10mm/sec CNT100;
   1:  PR[GP1:91,1] = PR[GP1:90,1] + -43.635;
   1:  PR[GP1:91,2] = PR[GP1:90,2] + -33.378;
   1:L PR[91] 10mm/sec CNT100;
   1:  PR[GP1:91,1] = PR[GP1:90,1] + -37.396;
   1:  PR[GP1:91,2] = PR[GP1:90,2] + -35.664;
   1:L PR[91] 10mm/sec CNT100;
   1:  PR[GP1:91,1] = PR[GP1:90,1] + -31.462;
   1:  PR[GP1:91,2] = PR[GP1:90,2] + -36.508;
   1:L PR[91] 10mm/sec CNT100;
   1:  PR[GP1:91,1] = PR[GP1:90,1] + -27.407;
   1:  PR[GP1:91,2] = PR[GP1:90,2] + -36.897;
   1:L PR[91] 10mm/sec CNT100;
   1:  PR[GP1:91,1] = PR[GP1:90,1] + -21.686;
   1:  PR[GP1:91,2] = PR[GP1:90,2] + -36.519;
   1:L PR[91] 10mm/sec CNT100;
   1:  PR[GP1:91,1] = PR[GP1:90,1] + -17.025;
   1:  PR[GP1:91,2] = PR[GP1:90,2] + -35.453;
   1:L PR[91] 10mm/sec CNT100;
   1:  PR[GP1:91,1] = PR[GP1:90,1] + -11.776;
   1:  PR[GP1:91,2] = PR[GP1:90,2] + -33.946;
   1:L PR[91] 10mm/sec CNT100;
   1:  PR[GP1:91,1] = PR[GP1:90,1] + -7.613;
   1:  PR[GP1:91,2] = PR[GP1:90,2] + -31.506;
   1:L PR[91] 10mm/sec CNT100;
   1:  PR[GP1:91,1] = PR[GP1:90,1] + -4.793;
   1:  PR[GP1:91,2] = PR[GP1:90,2] + -29.971;
   1:L PR[91] 10mm/sec CNT100;
   1:  PR[GP1:91,1] = PR[GP1:90,1] + -0.262;
   1:  PR[GP1:91,2] = PR[GP1:90,2] + -26.062;
   1:L PR[91] 10mm/sec CNT100;
   1:  PR[GP1:91,1] = PR[GP1:90,1] + 4.030;
   1:  PR[GP1:91,2] = PR[GP1:90,2] + -30.051;
   1:  PR[GP1:91,3] = PR[GP1:90,3] + 58.255;
   1:L PR[91] 10mm/sec CNT100;
   1:  PR[GP1:91,1] = PR[GP1:90,1] + 6.668;
   1:  PR[GP1:91,2] = PR[GP1:90,2] + -31.483;
   1:L PR[91] 10mm/sec CNT100;
   1:  PR[GP1:91,1] = PR[GP1:90,1] + 10.990;
   1:  PR[GP1:91,2] = PR[GP1:90,2] + -34.012;
   1:L PR[91] 10mm/sec CNT100;
   1:  PR[GP1:91,1] = PR[GP1:90,1] + 16.126;
   1:  PR[GP1:91,2] = PR[GP1:90,2] + -35.487;
   1:L PR[91] 10mm/sec CNT100;
   1:  PR[GP1:91,1] = PR[GP1:90,1] + 20.985;
   1:  PR[GP1:91,2] = PR[GP1:90,2] + -36.599;
   1:L PR[91] 10mm/sec CNT100;
   1:  PR[GP1:91,1] = PR[GP1:90,1] + 26.553;
   1:  PR[GP1:91,2] = PR[GP1:90,2] + -36.969;
   1:L PR[91] 10mm/sec CNT100;
   1:  PR[GP1:91,1] = PR[GP1:90,1] + 32.780;
   1:  PR[GP1:91,2] = PR[GP1:90,2] + -36.109;
   1:L PR[91] 10mm/sec CNT100;
   1:  PR[GP1:91,1] = PR[GP1:90,1] + 36.632;
   1:  PR[GP1:91,2] = PR[GP1:90,2] + -35.735;
   1:L PR[91] 10mm/sec CNT100;
   1:  PR[GP1:91,1] = PR[GP1:90,1] + 42.739;
   1:  PR[GP1:91,2] = PR[GP1:90,2] + -33.506;
   1:L PR[91] 10mm/sec CNT100;
   1:  PR[GP1:91,1] = PR[GP1:90,1] + 45.592;
   1:  PR[GP1:91,2] = PR[GP1:90,2] + -32.251;
   1:L PR[91] 10mm/sec CNT100;
   1:  PR[GP1:91,1] = PR[GP1:90,1] + 51.194;
   1:  PR[GP1:91,2] = PR[GP1:90,2] + -28.736;
   1:L PR[91] 10mm/sec CNT100;
   1:  PR[GP1:91,1] = PR[GP1:90,1] + 56.285;
   1:  PR[GP1:91,2] = PR[GP1:90,2] + -23.774;
   1:L PR[91] 10mm/sec CNT100;
   1:  PR[GP1:91,1] = PR[GP1:90,1] + 57.794;
   1:  PR[GP1:91,2] = PR[GP1:90,2] + -22.402;
   1:L PR[91] 10mm/sec CNT100;
   1:  PR[GP1:91,1] = PR[GP1:90,1] + 61.757;
   1:  PR[GP1:91,2] = PR[GP1:90,2] + -16.255;
   1:L PR[91] 10mm/sec CNT100;
   1:  PR[GP1:91,1] = PR[GP1:90,1] + 62.520;
   1:  PR[GP1:91,2] = PR[GP1:90,2] + -14.877;
   1:L PR[91] 10mm/sec CNT100;
   1:  PR[GP1:91,1] = PR[GP1:90,1] + 64.979;
   1:  PR[GP1:91,2] = PR[GP1:90,2] + -8.190;
   1:L PR[91] 10mm/sec CNT100;
   1:  PR[GP1:91,1] = PR[GP1:90,1] + 65.805;
   1:  PR[GP1:91,2] = PR[GP1:90,2] + -0.922;
   1:L PR[91] 10mm/sec CNT100;
   1:  PR[GP1:91,1] = PR[GP1:90,1] + 66.013;
   1:  PR[GP1:91,2] = PR[GP1:90,2] + 0.296;
   1:L PR[91] 10mm/sec CNT100;
   1:  PR[GP1:91,1] = PR[GP1:90,1] + 65.204;
   1:  PR[GP1:91,2] = PR[GP1:90,2] + 7.450;
   1:L PR[91] 10mm/sec CNT100;
   1:  PR[GP1:91,1] = PR[GP1:90,1] + 64.984;
   1:  PR[GP1:91,2] = PR[GP1:90,2] + 8.735;
   1:L PR[91] 10mm/sec CNT100;
   1:  PR[GP1:91,1] = PR[GP1:90,1] + 62.519;
   1:  PR[GP1:91,2] = PR[GP1:90,2] + 15.438;
   1:L PR[91] 10mm/sec CNT100;
   1:  PR[GP1:91,1] = PR[GP1:90,1] + 61.753;
   1:  PR[GP1:91,2] = PR[GP1:90,2] + 16.819;
   1:L PR[91] 10mm/sec CNT100;
   1:  PR[GP1:91,1] = PR[GP1:90,1] + 57.783;
   1:  PR[GP1:91,2] = PR[GP1:90,2] + 22.976;
   1:L PR[91] 10mm/sec CNT100;
   1:  PR[GP1:91,1] = PR[GP1:90,1] + 53.007;
   1:  PR[GP1:91,2] = PR[GP1:90,2] + 27.653;
   1:L PR[91] 10mm/sec CNT100;
   1:  PR[GP1:91,1] = PR[GP1:90,1] + 51.190;
   1:  PR[GP1:91,2] = PR[GP1:90,2] + 29.298;
   1:L PR[91] 10mm/sec CNT100;
   1:  PR[GP1:91,1] = PR[GP1:90,1] + 45.576;
   1:  PR[GP1:91,2] = PR[GP1:90,2] + 32.820;
   1:L PR[91] 10mm/sec CNT100;
   1:  PR[GP1:91,1] = PR[GP1:90,1] + 42.712;
   1:  PR[GP1:91,2] = PR[GP1:90,2] + 34.071;
   1:L PR[91] 10mm/sec CNT100;
   1:  PR[GP1:91,1] = PR[GP1:90,1] + 36.588;
   1:  PR[GP1:91,2] = PR[GP1:90,2] + 36.306;
   1:L PR[91] 10mm/sec CNT100;
   1:  PR[GP1:91,1] = PR[GP1:90,1] + 30.790;
   1:  PR[GP1:91,2] = PR[GP1:90,2] + 37.128;
   1:L PR[91] 10mm/sec CNT100;
   1:  PR[GP1:91,1] = PR[GP1:90,1] + 26.517;
   1:  PR[GP1:91,2] = PR[GP1:90,2] + 37.525;
   1:L PR[91] 10mm/sec CNT100;
   1:  PR[GP1:91,1] = PR[GP1:90,1] + 20.935;
   1:  PR[GP1:91,2] = PR[GP1:90,2] + 37.154;
   1:L PR[91] 10mm/sec CNT100;
   1:  PR[GP1:91,1] = PR[GP1:90,1] + 15.995;
   1:  PR[GP1:91,2] = PR[GP1:90,2] + 35.987;
   1:L PR[91] 10mm/sec CNT100;
   1:  PR[GP1:91,1] = PR[GP1:90,1] + 10.883;
   1:  PR[GP1:91,2] = PR[GP1:90,2] + 34.518;
   1:L PR[91] 10mm/sec CNT100;
   1:  PR[GP1:91,1] = PR[GP1:90,1] + 6.242;
   1:  PR[GP1:91,2] = PR[GP1:90,2] + 32.023;
   1:L PR[91] 10mm/sec CNT100;
   1:  PR[GP1:91,1] = PR[GP1:90,1] + -0.263;
   1:  PR[GP1:91,2] = PR[GP1:90,2] + 26.732;
   1:L PR[91] 10mm/sec CNT100;
   1:  PR[GP1:91,1] = PR[GP1:90,1] + -6.751;
   1:  PR[GP1:91,2] = PR[GP1:90,2] + 32.008;
   1:L PR[91] 10mm/sec CNT100;
   1:  PR[GP1:91,1] = PR[GP1:90,1] + -11.413;
   1:  PR[GP1:91,2] = PR[GP1:90,2] + 34.520;
   1:L PR[91] 10mm/sec CNT100;
   1:  PR[GP1:91,1] = PR[GP1:90,1] + -16.518;
   1:  PR[GP1:91,2] = PR[GP1:90,2] + 35.988;
   1:L PR[91] 10mm/sec CNT100;
   1:  PR[GP1:91,1] = PR[GP1:90,1] + -21.459;
   1:  PR[GP1:91,2] = PR[GP1:90,2] + 37.154;
   1:L PR[91] 10mm/sec CNT100;
   1:  PR[GP1:91,1] = PR[GP1:90,1] + -27.045;
   1:  PR[GP1:91,2] = PR[GP1:90,2] + 37.523;
   1:L PR[91] 10mm/sec CNT100;
   1:  PR[GP1:91,1] = PR[GP1:90,1] + -33.298;
   1:  PR[GP1:91,2] = PR[GP1:90,2] + 36.658;
   1:L PR[91] 10mm/sec CNT100;
   1:  PR[GP1:91,1] = PR[GP1:90,1] + -37.160;
   1:  PR[GP1:91,2] = PR[GP1:90,2] + 36.295;
   1:L PR[91] 10mm/sec CNT100;
   1:  PR[GP1:91,1] = PR[GP1:90,1] + -43.263;
   1:  PR[GP1:91,2] = PR[GP1:90,2] + 34.059;
   1:L PR[91] 10mm/sec CNT100;
   1:  PR[GP1:91,1] = PR[GP1:90,1] + -46.125;
   1:  PR[GP1:91,2] = PR[GP1:90,2] + 32.808;
   1:L PR[91] 10mm/sec CNT100;
   1:  PR[GP1:91,1] = PR[GP1:90,1] + -51.763;
   1:  PR[GP1:91,2] = PR[GP1:90,2] + 29.253;
   1:L PR[91] 10mm/sec CNT100;
   1:  PR[GP1:91,1] = PR[GP1:90,1] + -56.866;
   1:  PR[GP1:91,2] = PR[GP1:90,2] + 24.272;
   1:L PR[91] 10mm/sec CNT100;
   1:  PR[GP1:91,1] = PR[GP1:90,1] + -58.377;
   1:  PR[GP1:91,2] = PR[GP1:90,2] + 22.903;
   1:L PR[91] 10mm/sec CNT100;
   1:  PR[GP1:91,1] = PR[GP1:90,1] + -62.299;
   1:  PR[GP1:91,2] = PR[GP1:90,2] + 16.783;
   1:L PR[91] 10mm/sec CNT100;
   1:  PR[GP1:91,1] = PR[GP1:90,1] + -63.064;
   1:  PR[GP1:91,2] = PR[GP1:90,2] + 15.401;
   1:L PR[91] 10mm/sec CNT100;
   1:  PR[GP1:91,1] = PR[GP1:90,1] + -65.533;
   1:  PR[GP1:91,2] = PR[GP1:90,2] + 8.597;
   1:L PR[91] 10mm/sec CNT100;
   1:  PR[GP1:91,1] = PR[GP1:90,1] + -66.330;
   1:  PR[GP1:91,2] = PR[GP1:90,2] + 1.482;
   1:L PR[91] 10mm/sec CNT100;
   1:  PR[GP1:91,1] = PR[GP1:90,1] + -66.539;
   1:  PR[GP1:91,2] = PR[GP1:90,2] + 0.261;
   1:L PR[91] 10mm/sec CNT100;
   1:  PR[GP1:91,1] = PR[GP1:90,1] + -65.759;
   1:  PR[GP1:91,2] = PR[GP1:90,2] + -6.740;
   1:L PR[91] 10mm/sec CNT100;
   1:  PR[GP1:91,1] = PR[GP1:90,1] + -65.540;
   1:  PR[GP1:91,2] = PR[GP1:90,2] + -8.019;
   1:L PR[91] 10mm/sec CNT100;
   1:  PR[GP1:91,1] = PR[GP1:90,1] + -63.065;
   1:  PR[GP1:91,2] = PR[GP1:90,2] + -14.840;
   1:L PR[91] 10mm/sec CNT100;
   1:  PR[GP1:91,1] = PR[GP1:90,1] + -62.303;
   1:  PR[GP1:91,2] = PR[GP1:90,2] + -16.219;
   1:L PR[91] 10mm/sec CNT100;
   1:  PR[GP1:91,1] = PR[GP1:90,1] + -58.376;
   1:  PR[GP1:91,2] = PR[GP1:90,2] + -22.349;
   1:L PR[91] 10mm/sec CNT100;
   1:  PR[GP1:91,1] = PR[GP1:90,1] + -53.594;
   1:  PR[GP1:91,2] = PR[GP1:90,2] + -27.041;
   1:L PR[91] 10mm/sec CNT100;
   1:  PR[GP1:91,1] = PR[GP1:90,1] + -51.787;
   1:  PR[GP1:91,2] = PR[GP1:90,2] + -28.680;
   1:L PR[91] 10mm/sec CNT100;
   1:  PR[GP1:91,1] = PR[GP1:90,1] + -46.141;
   1:  PR[GP1:91,2] = PR[GP1:90,2] + -32.240;
   1:L PR[91] 10mm/sec CNT100;
   1:  PR[GP1:91,1] = PR[GP1:90,1] + -43.291;
   1:  PR[GP1:91,2] = PR[GP1:90,2] + -33.494;
   1:L PR[91] 10mm/sec CNT100;
   1:  PR[GP1:91,1] = PR[GP1:90,1] + -37.178;
   1:  PR[GP1:91,2] = PR[GP1:90,2] + -35.733;
   1:L PR[91] 10mm/sec CNT100;
   1:  PR[GP1:91,1] = PR[GP1:90,1] + -31.364;
   1:  PR[GP1:91,2] = PR[GP1:90,2] + -36.560;
   1:L PR[91] 10mm/sec CNT100;
   1:  PR[GP1:91,1] = PR[GP1:90,1] + -27.107;
   1:  PR[GP1:91,2] = PR[GP1:90,2] + -36.969;
   1:L PR[91] 10mm/sec CNT100;
   1:  PR[GP1:91,1] = PR[GP1:90,1] + -21.510;
   1:  PR[GP1:91,2] = PR[GP1:90,2] + -36.600;
   1:L PR[91] 10mm/sec CNT100;
   1:  PR[GP1:91,1] = PR[GP1:90,1] + -16.650;
   1:  PR[GP1:91,2] = PR[GP1:90,2] + -35.488;
   1:L PR[91] 10mm/sec CNT100;
   1:  PR[GP1:91,1] = PR[GP1:90,1] + -11.522;
   1:  PR[GP1:91,2] = PR[GP1:90,2] + -34.015;
   1:L PR[91] 10mm/sec CNT100;
   1:  PR[GP1:91,1] = PR[GP1:90,1] + -7.202;
   1:  PR[GP1:91,2] = PR[GP1:90,2] + -31.484;
   1:L PR[91] 10mm/sec CNT100;
   1:  PR[GP1:91,1] = PR[GP1:90,1] + -4.549;
   1:  PR[GP1:91,2] = PR[GP1:90,2] + -30.040;
   1:L PR[91] 10mm/sec CNT100;
   1:  PR[GP1:91,1] = PR[GP1:90,1] + -0.262;
   1:  PR[GP1:91,2] = PR[GP1:90,2] + -26.341;
   1:L PR[91] 10mm/sec CNT100;
   1:  PR[GP1:91,1] = PR[GP1:90,1] + 3.785;
   1:  PR[GP1:91,2] = PR[GP1:90,2] + -30.119;
   1:  PR[GP1:91,3] = PR[GP1:90,3] + 58.865;
   1:L PR[91] 10mm/sec CNT100;
   1:  PR[GP1:91,1] = PR[GP1:90,1] + 6.258;
   1:  PR[GP1:91,2] = PR[GP1:90,2] + -31.461;
   1:L PR[91] 10mm/sec CNT100;
   1:  PR[GP1:91,1] = PR[GP1:90,1] + 10.736;
   1:  PR[GP1:91,2] = PR[GP1:90,2] + -34.082;
   1:L PR[91] 10mm/sec CNT100;
   1:  PR[GP1:91,1] = PR[GP1:90,1] + 15.750;
   1:  PR[GP1:91,2] = PR[GP1:90,2] + -35.522;
   1:L PR[91] 10mm/sec CNT100;
   1:  PR[GP1:91,1] = PR[GP1:90,1] + 20.808;
   1:  PR[GP1:91,2] = PR[GP1:90,2] + -36.679;
   1:L PR[91] 10mm/sec CNT100;
   1:  PR[GP1:91,1] = PR[GP1:90,1] + 26.253;
   1:  PR[GP1:91,2] = PR[GP1:90,2] + -37.041;
   1:L PR[91] 10mm/sec CNT100;
   1:  PR[GP1:91,1] = PR[GP1:90,1] + 32.344;
   1:  PR[GP1:91,2] = PR[GP1:90,2] + -36.200;
   1:L PR[91] 10mm/sec CNT100;
   1:  PR[GP1:91,1] = PR[GP1:90,1] + 36.414;
   1:  PR[GP1:91,2] = PR[GP1:90,2] + -35.805;
   1:L PR[91] 10mm/sec CNT100;
   1:  PR[GP1:91,1] = PR[GP1:90,1] + 42.395;
   1:  PR[GP1:91,2] = PR[GP1:90,2] + -33.622;
   1:L PR[91] 10mm/sec CNT100;
   1:  PR[GP1:91,1] = PR[GP1:90,1] + 45.447;
   1:  PR[GP1:91,2] = PR[GP1:90,2] + -32.280;
   1:L PR[91] 10mm/sec CNT100;
   1:  PR[GP1:91,1] = PR[GP1:90,1] + 50.939;
   1:  PR[GP1:91,2] = PR[GP1:90,2] + -28.834;
   1:L PR[91] 10mm/sec CNT100;
   1:  PR[GP1:91,1] = PR[GP1:90,1] + 55.930;
   1:  PR[GP1:91,2] = PR[GP1:90,2] + -23.969;
   1:L PR[91] 10mm/sec CNT100;
   1:  PR[GP1:91,1] = PR[GP1:90,1] + 57.607;
   1:  PR[GP1:91,2] = PR[GP1:90,2] + -22.443;
   1:L PR[91] 10mm/sec CNT100;
   1:  PR[GP1:91,1] = PR[GP1:90,1] + 61.495;
   1:  PR[GP1:91,2] = PR[GP1:90,2] + -16.413;
   1:L PR[91] 10mm/sec CNT100;
   1:  PR[GP1:91,1] = PR[GP1:90,1] + 62.366;
   1:  PR[GP1:91,2] = PR[GP1:90,2] + -14.840;
   1:L PR[91] 10mm/sec CNT100;
   1:  PR[GP1:91,1] = PR[GP1:90,1] + 64.779;
   1:  PR[GP1:91,2] = PR[GP1:90,2] + -8.277;
   1:L PR[91] 10mm/sec CNT100;
   1:  PR[GP1:91,1] = PR[GP1:90,1] + 65.590;
   1:  PR[GP1:91,2] = PR[GP1:90,2] + -1.142;
   1:L PR[91] 10mm/sec CNT100;
   1:  PR[GP1:91,1] = PR[GP1:90,1] + 65.835;
   1:  PR[GP1:91,2] = PR[GP1:90,2] + 0.296;
   1:L PR[91] 10mm/sec CNT100;
   1:  PR[GP1:91,1] = PR[GP1:90,1] + 65.041;
   1:  PR[GP1:91,2] = PR[GP1:90,2] + 7.319;
   1:L PR[91] 10mm/sec CNT100;
   1:  PR[GP1:91,1] = PR[GP1:90,1] + 64.784;
   1:  PR[GP1:91,2] = PR[GP1:90,2] + 8.822;
   1:L PR[91] 10mm/sec CNT100;
   1:  PR[GP1:91,1] = PR[GP1:90,1] + 62.364;
   1:  PR[GP1:91,2] = PR[GP1:90,2] + 15.401;
   1:L PR[91] 10mm/sec CNT100;
   1:  PR[GP1:91,1] = PR[GP1:90,1] + 61.490;
   1:  PR[GP1:91,2] = PR[GP1:90,2] + 16.977;
   1:L PR[91] 10mm/sec CNT100;
   1:  PR[GP1:91,1] = PR[GP1:90,1] + 57.595;
   1:  PR[GP1:91,2] = PR[GP1:90,2] + 23.018;
   1:L PR[91] 10mm/sec CNT100;
   1:  PR[GP1:91,1] = PR[GP1:90,1] + 52.909;
   1:  PR[GP1:91,2] = PR[GP1:90,2] + 27.607;
   1:L PR[91] 10mm/sec CNT100;
   1:  PR[GP1:91,1] = PR[GP1:90,1] + 50.933;
   1:  PR[GP1:91,2] = PR[GP1:90,2] + 29.396;
   1:L PR[91] 10mm/sec CNT100;
   1:  PR[GP1:91,1] = PR[GP1:90,1] + 45.430;
   1:  PR[GP1:91,2] = PR[GP1:90,2] + 32.849;
   1:L PR[91] 10mm/sec CNT100;
   1:  PR[GP1:91,1] = PR[GP1:90,1] + 42.366;
   1:  PR[GP1:91,2] = PR[GP1:90,2] + 34.187;
   1:L PR[91] 10mm/sec CNT100;
   1:  PR[GP1:91,1] = PR[GP1:90,1] + 36.369;
   1:  PR[GP1:91,2] = PR[GP1:90,2] + 36.376;
   1:L PR[91] 10mm/sec CNT100;
   1:  PR[GP1:91,1] = PR[GP1:90,1] + 30.691;
   1:  PR[GP1:91,2] = PR[GP1:90,2] + 37.181;
   1:L PR[91] 10mm/sec CNT100;
   1:  PR[GP1:91,1] = PR[GP1:90,1] + 26.215;
   1:  PR[GP1:91,2] = PR[GP1:90,2] + 37.597;
   1:L PR[91] 10mm/sec CNT100;
   1:  PR[GP1:91,1] = PR[GP1:90,1] + 20.756;
   1:  PR[GP1:91,2] = PR[GP1:90,2] + 37.234;
   1:L PR[91] 10mm/sec CNT100;
   1:  PR[GP1:91,1] = PR[GP1:90,1] + 15.614;
   1:  PR[GP1:91,2] = PR[GP1:90,2] + 36.020;
   1:L PR[91] 10mm/sec CNT100;
   1:  PR[GP1:91,1] = PR[GP1:90,1] + 10.625;
   1:  PR[GP1:91,2] = PR[GP1:90,2] + 34.585;
   1:L PR[91] 10mm/sec CNT100;
   1:  PR[GP1:91,1] = PR[GP1:90,1] + 6.069;
   1:  PR[GP1:91,2] = PR[GP1:90,2] + 32.138;
   1:L PR[91] 10mm/sec CNT100;
   1:  PR[GP1:91,1] = PR[GP1:90,1] + -0.263;
   1:  PR[GP1:91,2] = PR[GP1:90,2] + 26.987;
   1:L PR[91] 10mm/sec CNT100;
   1:  PR[GP1:91,1] = PR[GP1:90,1] + -6.579;
   1:  PR[GP1:91,2] = PR[GP1:90,2] + 32.122;
   1:L PR[91] 10mm/sec CNT100;
   1:  PR[GP1:91,1] = PR[GP1:90,1] + -11.154;
   1:  PR[GP1:91,2] = PR[GP1:90,2] + 34.588;
   1:L PR[91] 10mm/sec CNT100;
   1:  PR[GP1:91,1] = PR[GP1:90,1] + -16.137;
   1:  PR[GP1:91,2] = PR[GP1:90,2] + 36.020;
   1:L PR[91] 10mm/sec CNT100;
   1:  PR[GP1:91,1] = PR[GP1:90,1] + -21.280;
   1:  PR[GP1:91,2] = PR[GP1:90,2] + 37.234;
   1:L PR[91] 10mm/sec CNT100;
   1:  PR[GP1:91,1] = PR[GP1:90,1] + -26.742;
   1:  PR[GP1:91,2] = PR[GP1:90,2] + 37.595;
   1:L PR[91] 10mm/sec CNT100;
   1:  PR[GP1:91,1] = PR[GP1:90,1] + -32.858;
   1:  PR[GP1:91,2] = PR[GP1:90,2] + 36.748;
   1:L PR[91] 10mm/sec CNT100;
   1:  PR[GP1:91,1] = PR[GP1:90,1] + -36.940;
   1:  PR[GP1:91,2] = PR[GP1:90,2] + 36.365;
   1:L PR[91] 10mm/sec CNT100;
   1:  PR[GP1:91,1] = PR[GP1:90,1] + -42.917;
   1:  PR[GP1:91,2] = PR[GP1:90,2] + 34.176;
   1:L PR[91] 10mm/sec CNT100;
   1:  PR[GP1:91,1] = PR[GP1:90,1] + -45.978;
   1:  PR[GP1:91,2] = PR[GP1:90,2] + 32.837;
   1:L PR[91] 10mm/sec CNT100;
   1:  PR[GP1:91,1] = PR[GP1:90,1] + -51.505;
   1:  PR[GP1:91,2] = PR[GP1:90,2] + 29.352;
   1:L PR[91] 10mm/sec CNT100;
   1:  PR[GP1:91,1] = PR[GP1:90,1] + -56.509;
   1:  PR[GP1:91,2] = PR[GP1:90,2] + 24.468;
   1:L PR[91] 10mm/sec CNT100;
   1:  PR[GP1:91,1] = PR[GP1:90,1] + -58.189;
   1:  PR[GP1:91,2] = PR[GP1:90,2] + 22.947;
   1:L PR[91] 10mm/sec CNT100;
   1:  PR[GP1:91,1] = PR[GP1:90,1] + -62.036;
   1:  PR[GP1:91,2] = PR[GP1:90,2] + 16.942;
   1:L PR[91] 10mm/sec CNT100;
   1:  PR[GP1:91,1] = PR[GP1:90,1] + -62.909;
   1:  PR[GP1:91,2] = PR[GP1:90,2] + 15.365;
   1:L PR[91] 10mm/sec CNT100;
   1:  PR[GP1:91,1] = PR[GP1:90,1] + -65.333;
   1:  PR[GP1:91,2] = PR[GP1:90,2] + 8.686;
   1:L PR[91] 10mm/sec CNT100;
   1:  PR[GP1:91,1] = PR[GP1:90,1] + -66.115;
   1:  PR[GP1:91,2] = PR[GP1:90,2] + 1.702;
   1:L PR[91] 10mm/sec CNT100;
   1:  PR[GP1:91,1] = PR[GP1:90,1] + -66.362;
   1:  PR[GP1:91,2] = PR[GP1:90,2] + 0.261;
   1:L PR[91] 10mm/sec CNT100;
   1:  PR[GP1:91,1] = PR[GP1:90,1] + -65.596;
   1:  PR[GP1:91,2] = PR[GP1:90,2] + -6.613;
   1:L PR[91] 10mm/sec CNT100;
   1:  PR[GP1:91,1] = PR[GP1:90,1] + -65.340;
   1:  PR[GP1:91,2] = PR[GP1:90,2] + -8.109;
   1:L PR[91] 10mm/sec CNT100;
   1:  PR[GP1:91,1] = PR[GP1:90,1] + -62.910;
   1:  PR[GP1:91,2] = PR[GP1:90,2] + -14.804;
   1:L PR[91] 10mm/sec CNT100;
   1:  PR[GP1:91,1] = PR[GP1:90,1] + -62.041;
   1:  PR[GP1:91,2] = PR[GP1:90,2] + -16.378;
   1:L PR[91] 10mm/sec CNT100;
   1:  PR[GP1:91,1] = PR[GP1:90,1] + -58.188;
   1:  PR[GP1:91,2] = PR[GP1:90,2] + -22.392;
   1:L PR[91] 10mm/sec CNT100;
   1:  PR[GP1:91,1] = PR[GP1:90,1] + -53.496;
   1:  PR[GP1:91,2] = PR[GP1:90,2] + -26.995;
   1:L PR[91] 10mm/sec CNT100;
   1:  PR[GP1:91,1] = PR[GP1:90,1] + -51.530;
   1:  PR[GP1:91,2] = PR[GP1:90,2] + -28.778;
   1:L PR[91] 10mm/sec CNT100;
   1:  PR[GP1:91,1] = PR[GP1:90,1] + -45.995;
   1:  PR[GP1:91,2] = PR[GP1:90,2] + -32.268;
   1:L PR[91] 10mm/sec CNT100;
   1:  PR[GP1:91,1] = PR[GP1:90,1] + -42.946;
   1:  PR[GP1:91,2] = PR[GP1:90,2] + -33.610;
   1:L PR[91] 10mm/sec CNT100;
   1:  PR[GP1:91,1] = PR[GP1:90,1] + -36.960;
   1:  PR[GP1:91,2] = PR[GP1:90,2] + -35.803;
   1:L PR[91] 10mm/sec CNT100;
   1:  PR[GP1:91,1] = PR[GP1:90,1] + -31.266;
   1:  PR[GP1:91,2] = PR[GP1:90,2] + -36.613;
   1:L PR[91] 10mm/sec CNT100;
   1:  PR[GP1:91,1] = PR[GP1:90,1] + -26.806;
   1:  PR[GP1:91,2] = PR[GP1:90,2] + -37.041;
   1:L PR[91] 10mm/sec CNT100;
   1:  PR[GP1:91,1] = PR[GP1:90,1] + -21.333;
   1:  PR[GP1:91,2] = PR[GP1:90,2] + -36.680;
   1:L PR[91] 10mm/sec CNT100;
   1:  PR[GP1:91,1] = PR[GP1:90,1] + -16.275;
   1:  PR[GP1:91,2] = PR[GP1:90,2] + -35.522;
   1:L PR[91] 10mm/sec CNT100;
   1:  PR[GP1:91,1] = PR[GP1:90,1] + -11.267;
   1:  PR[GP1:91,2] = PR[GP1:90,2] + -34.084;
   1:L PR[91] 10mm/sec CNT100;
   1:  PR[GP1:91,1] = PR[GP1:90,1] + -6.792;
   1:  PR[GP1:91,2] = PR[GP1:90,2] + -31.463;
   1:L PR[91] 10mm/sec CNT100;
   1:  PR[GP1:91,1] = PR[GP1:90,1] + -4.305;
   1:  PR[GP1:91,2] = PR[GP1:90,2] + -30.109;
   1:L PR[91] 10mm/sec CNT100;
   1:  PR[GP1:91,1] = PR[GP1:90,1] + -0.263;
   1:  PR[GP1:91,2] = PR[GP1:90,2] + -26.620;
   1:L PR[91] 10mm/sec CNT100;
   1:  PR[GP1:91,1] = PR[GP1:90,1] + 3.541;
   1:  PR[GP1:91,2] = PR[GP1:90,2] + -30.187;
   1:  PR[GP1:91,3] = PR[GP1:90,3] + 59.475;
   1:L PR[91] 10mm/sec CNT100;
   1:  PR[GP1:91,1] = PR[GP1:90,1] + 5.847;
   1:  PR[GP1:91,2] = PR[GP1:90,2] + -31.439;
   1:L PR[91] 10mm/sec CNT100;
   1:  PR[GP1:91,1] = PR[GP1:90,1] + 10.481;
   1:  PR[GP1:91,2] = PR[GP1:90,2] + -34.151;
   1:L PR[91] 10mm/sec CNT100;
   1:  PR[GP1:91,1] = PR[GP1:90,1] + 15.375;
   1:  PR[GP1:91,2] = PR[GP1:90,2] + -35.557;
   1:L PR[91] 10mm/sec CNT100;
   1:  PR[GP1:91,1] = PR[GP1:90,1] + 20.632;
   1:  PR[GP1:91,2] = PR[GP1:90,2] + -36.760;
   1:L PR[91] 10mm/sec CNT100;
   1:  PR[GP1:91,1] = PR[GP1:90,1] + 25.953;
   1:  PR[GP1:91,2] = PR[GP1:90,2] + -37.113;
   1:L PR[91] 10mm/sec CNT100;
   1:  PR[GP1:91,1] = PR[GP1:90,1] + 31.907;
   1:  PR[GP1:91,2] = PR[GP1:90,2] + -36.291;
   1:L PR[91] 10mm/sec CNT100;
   1:  PR[GP1:91,1] = PR[GP1:90,1] + 36.197;
   1:  PR[GP1:91,2] = PR[GP1:90,2] + -35.874;
   1:L PR[91] 10mm/sec CNT100;
   1:  PR[GP1:91,1] = PR[GP1:90,1] + 42.051;
   1:  PR[GP1:91,2] = PR[GP1:90,2] + -33.737;
   1:L PR[91] 10mm/sec CNT100;
   1:  PR[GP1:91,1] = PR[GP1:90,1] + 45.301;
   1:  PR[GP1:91,2] = PR[GP1:90,2] + -32.308;
   1:L PR[91] 10mm/sec CNT100;
   1:  PR[GP1:91,1] = PR[GP1:90,1] + 50.683;
   1:  PR[GP1:91,2] = PR[GP1:90,2] + -28.931;
   1:L PR[91] 10mm/sec CNT100;
   1:  PR[GP1:91,1] = PR[GP1:90,1] + 55.575;
   1:  PR[GP1:91,2] = PR[GP1:90,2] + -24.163;
   1:L PR[91] 10mm/sec CNT100;
   1:  PR[GP1:91,1] = PR[GP1:90,1] + 57.420;
   1:  PR[GP1:91,2] = PR[GP1:90,2] + -22.485;
   1:L PR[91] 10mm/sec CNT100;
   1:  PR[GP1:91,1] = PR[GP1:90,1] + 61.234;
   1:  PR[GP1:91,2] = PR[GP1:90,2] + -16.570;
   1:L PR[91] 10mm/sec CNT100;
   1:  PR[GP1:91,1] = PR[GP1:90,1] + 62.211;
   1:  PR[GP1:91,2] = PR[GP1:90,2] + -14.803;
   1:L PR[91] 10mm/sec CNT100;
   1:  PR[GP1:91,1] = PR[GP1:90,1] + 64.580;
   1:  PR[GP1:91,2] = PR[GP1:90,2] + -8.363;
   1:L PR[91] 10mm/sec CNT100;
   1:  PR[GP1:91,1] = PR[GP1:90,1] + 65.376;
   1:  PR[GP1:91,2] = PR[GP1:90,2] + -1.362;
   1:L PR[91] 10mm/sec CNT100;
   1:  PR[GP1:91,1] = PR[GP1:90,1] + 65.658;
   1:  PR[GP1:91,2] = PR[GP1:90,2] + 0.296;
   1:L PR[91] 10mm/sec CNT100;
   1:  PR[GP1:91,1] = PR[GP1:90,1] + 64.879;
   1:  PR[GP1:91,2] = PR[GP1:90,2] + 7.189;
   1:L PR[91] 10mm/sec CNT100;
   1:  PR[GP1:91,1] = PR[GP1:90,1] + 64.584;
   1:  PR[GP1:91,2] = PR[GP1:90,2] + 8.909;
   1:L PR[91] 10mm/sec CNT100;
   1:  PR[GP1:91,1] = PR[GP1:90,1] + 62.210;
   1:  PR[GP1:91,2] = PR[GP1:90,2] + 15.365;
   1:L PR[91] 10mm/sec CNT100;
   1:  PR[GP1:91,1] = PR[GP1:90,1] + 61.228;
   1:  PR[GP1:91,2] = PR[GP1:90,2] + 17.135;
   1:L PR[91] 10mm/sec CNT100;
   1:  PR[GP1:91,1] = PR[GP1:90,1] + 57.408;
   1:  PR[GP1:91,2] = PR[GP1:90,2] + 23.061;
   1:L PR[91] 10mm/sec CNT100;
   1:  PR[GP1:91,1] = PR[GP1:90,1] + 52.812;
   1:  PR[GP1:91,2] = PR[GP1:90,2] + 27.561;
   1:L PR[91] 10mm/sec CNT100;
   1:  PR[GP1:91,1] = PR[GP1:90,1] + 50.676;
   1:  PR[GP1:91,2] = PR[GP1:90,2] + 29.494;
   1:L PR[91] 10mm/sec CNT100;
   1:  PR[GP1:91,1] = PR[GP1:90,1] + 45.283;
   1:  PR[GP1:91,2] = PR[GP1:90,2] + 32.878;
   1:L PR[91] 10mm/sec CNT100;
   1:  PR[GP1:91,1] = PR[GP1:90,1] + 42.020;
   1:  PR[GP1:91,2] = PR[GP1:90,2] + 34.303;
   1:L PR[91] 10mm/sec CNT100;
   1:  PR[GP1:91,1] = PR[GP1:90,1] + 36.149;
   1:  PR[GP1:91,2] = PR[GP1:90,2] + 36.446;
   1:L PR[91] 10mm/sec CNT100;
   1:  PR[GP1:91,1] = PR[GP1:90,1] + 30.591;
   1:  PR[GP1:91,2] = PR[GP1:90,2] + 37.234;
   1:L PR[91] 10mm/sec CNT100;
   1:  PR[GP1:91,1] = PR[GP1:90,1] + 25.913;
   1:  PR[GP1:91,2] = PR[GP1:90,2] + 37.669;
   1:L PR[91] 10mm/sec CNT100;
   1:  PR[GP1:91,1] = PR[GP1:90,1] + 20.577;
   1:  PR[GP1:91,2] = PR[GP1:90,2] + 37.314;
   1:L PR[91] 10mm/sec CNT100;
   1:  PR[GP1:91,1] = PR[GP1:90,1] + 15.234;
   1:  PR[GP1:91,2] = PR[GP1:90,2] + 36.052;
   1:L PR[91] 10mm/sec CNT100;
   1:  PR[GP1:91,1] = PR[GP1:90,1] + 10.367;
   1:  PR[GP1:91,2] = PR[GP1:90,2] + 34.653;
   1:L PR[91] 10mm/sec CNT100;
   1:  PR[GP1:91,1] = PR[GP1:90,1] + 5.897;
   1:  PR[GP1:91,2] = PR[GP1:90,2] + 32.252;
   1:L PR[91] 10mm/sec CNT100;
   1:  PR[GP1:91,1] = PR[GP1:90,1] + -0.263;
   1:  PR[GP1:91,2] = PR[GP1:90,2] + 27.242;
   1:L PR[91] 10mm/sec CNT100;
   1:  PR[GP1:91,1] = PR[GP1:90,1] + -6.406;
   1:  PR[GP1:91,2] = PR[GP1:90,2] + 32.237;
   1:L PR[91] 10mm/sec CNT100;
   1:  PR[GP1:91,1] = PR[GP1:90,1] + -10.896;
   1:  PR[GP1:91,2] = PR[GP1:90,2] + 34.655;
   1:L PR[91] 10mm/sec CNT100;
   1:  PR[GP1:91,1] = PR[GP1:90,1] + -15.756;
   1:  PR[GP1:91,2] = PR[GP1:90,2] + 36.053;
   1:L PR[91] 10mm/sec CNT100;
   1:  PR[GP1:91,1] = PR[GP1:90,1] + -21.101;
   1:  PR[GP1:91,2] = PR[GP1:90,2] + 37.314;
   1:L PR[91] 10mm/sec CNT100;
   1:  PR[GP1:91,1] = PR[GP1:90,1] + -26.440;
   1:  PR[GP1:91,2] = PR[GP1:90,2] + 37.667;
   1:L PR[91] 10mm/sec CNT100;
   1:  PR[GP1:91,1] = PR[GP1:90,1] + -32.419;
   1:  PR[GP1:91,2] = PR[GP1:90,2] + 36.839;
   1:L PR[91] 10mm/sec CNT100;
   1:  PR[GP1:91,1] = PR[GP1:90,1] + -36.720;
   1:  PR[GP1:91,2] = PR[GP1:90,2] + 36.435;
   1:L PR[91] 10mm/sec CNT100;
   1:  PR[GP1:91,1] = PR[GP1:90,1] + -42.570;
   1:  PR[GP1:91,2] = PR[GP1:90,2] + 34.292;
   1:L PR[91] 10mm/sec CNT100;
   1:  PR[GP1:91,1] = PR[GP1:90,1] + -45.832;
   1:  PR[GP1:91,2] = PR[GP1:90,2] + 32.866;
   1:L PR[91] 10mm/sec CNT100;
   1:  PR[GP1:91,1] = PR[GP1:90,1] + -51.248;
   1:  PR[GP1:91,2] = PR[GP1:90,2] + 29.451;
   1:L PR[91] 10mm/sec CNT100;
   1:  PR[GP1:91,1] = PR[GP1:90,1] + -56.151;
   1:  PR[GP1:91,2] = PR[GP1:90,2] + 24.665;
   1:L PR[91] 10mm/sec CNT100;
   1:  PR[GP1:91,1] = PR[GP1:90,1] + -58.000;
   1:  PR[GP1:91,2] = PR[GP1:90,2] + 22.991;
   1:L PR[91] 10mm/sec CNT100;
   1:  PR[GP1:91,1] = PR[GP1:90,1] + -61.773;
   1:  PR[GP1:91,2] = PR[GP1:90,2] + 17.101;
   1:L PR[91] 10mm/sec CNT100;
   1:  PR[GP1:91,1] = PR[GP1:90,1] + -62.754;
   1:  PR[GP1:91,2] = PR[GP1:90,2] + 15.329;
   1:L PR[91] 10mm/sec CNT100;
   1:  PR[GP1:91,1] = PR[GP1:90,1] + -65.133;
   1:  PR[GP1:91,2] = PR[GP1:90,2] + 8.776;
   1:L PR[91] 10mm/sec CNT100;
   1:  PR[GP1:91,1] = PR[GP1:90,1] + -65.901;
   1:  PR[GP1:91,2] = PR[GP1:90,2] + 1.922;
   1:L PR[91] 10mm/sec CNT100;
   1:  PR[GP1:91,1] = PR[GP1:90,1] + -66.185;
   1:  PR[GP1:91,2] = PR[GP1:90,2] + 0.261;
   1:L PR[91] 10mm/sec CNT100;
   1:  PR[GP1:91,1] = PR[GP1:90,1] + -65.433;
   1:  PR[GP1:91,2] = PR[GP1:90,2] + -6.485;
   1:L PR[91] 10mm/sec CNT100;
   1:  PR[GP1:91,1] = PR[GP1:90,1] + -65.140;
   1:  PR[GP1:91,2] = PR[GP1:90,2] + -8.198;
   1:L PR[91] 10mm/sec CNT100;
   1:  PR[GP1:91,1] = PR[GP1:90,1] + -62.756;
   1:  PR[GP1:91,2] = PR[GP1:90,2] + -14.767;
   1:L PR[91] 10mm/sec CNT100;
   1:  PR[GP1:91,1] = PR[GP1:90,1] + -61.779;
   1:  PR[GP1:91,2] = PR[GP1:90,2] + -16.536;
   1:L PR[91] 10mm/sec CNT100;
   1:  PR[GP1:91,1] = PR[GP1:90,1] + -58.000;
   1:  PR[GP1:91,2] = PR[GP1:90,2] + -22.434;
   1:L PR[91] 10mm/sec CNT100;
   1:  PR[GP1:91,1] = PR[GP1:90,1] + -53.398;
   1:  PR[GP1:91,2] = PR[GP1:90,2] + -26.949;
   1:L PR[91] 10mm/sec CNT100;
   1:  PR[GP1:91,1] = PR[GP1:90,1] + -51.274;
   1:  PR[GP1:91,2] = PR[GP1:90,2] + -28.877;
   1:L PR[91] 10mm/sec CNT100;
   1:  PR[GP1:91,1] = PR[GP1:90,1] + -45.850;
   1:  PR[GP1:91,2] = PR[GP1:90,2] + -32.296;
   1:L PR[91] 10mm/sec CNT100;
   1:  PR[GP1:91,1] = PR[GP1:90,1] + -42.601;
   1:  PR[GP1:91,2] = PR[GP1:90,2] + -33.726;
   1:L PR[91] 10mm/sec CNT100;
   1:  PR[GP1:91,1] = PR[GP1:90,1] + -36.741;
   1:  PR[GP1:91,2] = PR[GP1:90,2] + -35.873;
   1:L PR[91] 10mm/sec CNT100;
   1:  PR[GP1:91,1] = PR[GP1:90,1] + -31.169;
   1:  PR[GP1:91,2] = PR[GP1:90,2] + -36.666;
   1:L PR[91] 10mm/sec CNT100;
   1:  PR[GP1:91,1] = PR[GP1:90,1] + -26.506;
   1:  PR[GP1:91,2] = PR[GP1:90,2] + -37.113;
   1:L PR[91] 10mm/sec CNT100;
   1:  PR[GP1:91,1] = PR[GP1:90,1] + -21.156;
   1:  PR[GP1:91,2] = PR[GP1:90,2] + -36.760;
   1:L PR[91] 10mm/sec CNT100;
   1:  PR[GP1:91,1] = PR[GP1:90,1] + -15.899;
   1:  PR[GP1:91,2] = PR[GP1:90,2] + -35.557;
   1:L PR[91] 10mm/sec CNT100;
   1:  PR[GP1:91,1] = PR[GP1:90,1] + -11.012;
   1:  PR[GP1:91,2] = PR[GP1:90,2] + -34.154;
   1:L PR[91] 10mm/sec CNT100;
   1:  PR[GP1:91,1] = PR[GP1:90,1] + -6.381;
   1:  PR[GP1:91,2] = PR[GP1:90,2] + -31.441;
   1:L PR[91] 10mm/sec CNT100;
   1:  PR[GP1:91,1] = PR[GP1:90,1] + -4.062;
   1:  PR[GP1:91,2] = PR[GP1:90,2] + -30.178;
   1:L PR[91] 10mm/sec CNT100;
   1:  PR[GP1:91,1] = PR[GP1:90,1] + -0.263;
   1:  PR[GP1:91,2] = PR[GP1:90,2] + -26.900;
   1:L PR[91] 10mm/sec CNT100;
   1:  PR[GP1:91,1] = PR[GP1:90,1] + 3.297;
   1:  PR[GP1:91,2] = PR[GP1:90,2] + -30.256;
   1:  PR[GP1:91,3] = PR[GP1:90,3] + 60.085;
   1:L PR[91] 10mm/sec CNT100;
   1:  PR[GP1:91,1] = PR[GP1:90,1] + 5.437;
   1:  PR[GP1:91,2] = PR[GP1:90,2] + -31.417;
   1:L PR[91] 10mm/sec CNT100;
   1:  PR[GP1:91,1] = PR[GP1:90,1] + 10.226;
   1:  PR[GP1:91,2] = PR[GP1:90,2] + -34.221;
   1:L PR[91] 10mm/sec CNT100;
   1:  PR[GP1:91,1] = PR[GP1:90,1] + 15.000;
   1:  PR[GP1:91,2] = PR[GP1:90,2] + -35.592;
   1:L PR[91] 10mm/sec CNT100;
   1:  PR[GP1:91,1] = PR[GP1:90,1] + 20.455;
   1:  PR[GP1:91,2] = PR[GP1:90,2] + -36.840;
   1:L PR[91] 10mm/sec CNT100;
   1:  PR[GP1:91,1] = PR[GP1:90,1] + 25.653;
   1:  PR[GP1:91,2] = PR[GP1:90,2] + -37.185;
   1:L PR[91] 10mm/sec CNT100;
   1:  PR[GP1:91,1] = PR[GP1:90,1] + 31.471;
   1:  PR[GP1:91,2] = PR[GP1:90,2] + -36.382;
   1:L PR[91] 10mm/sec CNT100;
   1:  PR[GP1:91,1] = PR[GP1:90,1] + 35.979;
   1:  PR[GP1:91,2] = PR[GP1:90,2] + -35.944;
   1:L PR[91] 10mm/sec CNT100;
   1:  PR[GP1:91,1] = PR[GP1:90,1] + 41.707;
   1:  PR[GP1:91,2] = PR[GP1:90,2] + -33.853;
   1:L PR[91] 10mm/sec CNT100;
   1:  PR[GP1:91,1] = PR[GP1:90,1] + 45.156;
   1:  PR[GP1:91,2] = PR[GP1:90,2] + -32.336;
   1:L PR[91] 10mm/sec CNT100;
   1:  PR[GP1:91,1] = PR[GP1:90,1] + 50.428;
   1:  PR[GP1:91,2] = PR[GP1:90,2] + -29.029;
   1:L PR[91] 10mm/sec CNT100;
   1:  PR[GP1:91,1] = PR[GP1:90,1] + 55.220;
   1:  PR[GP1:91,2] = PR[GP1:90,2] + -24.358;
   1:L PR[91] 10mm/sec CNT100;
   1:  PR[GP1:91,1] = PR[GP1:90,1] + 57.233;
   1:  PR[GP1:91,2] = PR[GP1:90,2] + -22.526;
   1:L PR[91] 10mm/sec CNT100;
   1:  PR[GP1:91,1] = PR[GP1:90,1] + 60.972;
   1:  PR[GP1:91,2] = PR[GP1:90,2] + -16.728;
   1:L PR[91] 10mm/sec CNT100;
   1:  PR[GP1:91,1] = PR[GP1:90,1] + 62.057;
   1:  PR[GP1:91,2] = PR[GP1:90,2] + -14.766;
   1:L PR[91] 10mm/sec CNT100;
   1:  PR[GP1:91,1] = PR[GP1:90,1] + 64.380;
   1:  PR[GP1:91,2] = PR[GP1:90,2] + -8.450;
   1:L PR[91] 10mm/sec CNT100;
   1:  PR[GP1:91,1] = PR[GP1:90,1] + 65.161;
   1:  PR[GP1:91,2] = PR[GP1:90,2] + -1.581;
   1:L PR[91] 10mm/sec CNT100;
   1:  PR[GP1:91,1] = PR[GP1:90,1] + 65.481;
   1:  PR[GP1:91,2] = PR[GP1:90,2] + 0.296;
   1:L PR[91] 10mm/sec CNT100;
   1:  PR[GP1:91,1] = PR[GP1:90,1] + 64.716;
   1:  PR[GP1:91,2] = PR[GP1:90,2] + 7.058;
   1:L PR[91] 10mm/sec CNT100;
   1:  PR[GP1:91,1] = PR[GP1:90,1] + 64.385;
   1:  PR[GP1:91,2] = PR[GP1:90,2] + 8.996;
   1:L PR[91] 10mm/sec CNT100;
   1:  PR[GP1:91,1] = PR[GP1:90,1] + 62.056;
   1:  PR[GP1:91,2] = PR[GP1:90,2] + 15.328;
   1:L PR[91] 10mm/sec CNT100;
   1:  PR[GP1:91,1] = PR[GP1:90,1] + 60.966;
   1:  PR[GP1:91,2] = PR[GP1:90,2] + 17.294;
   1:L PR[91] 10mm/sec CNT100;
   1:  PR[GP1:91,1] = PR[GP1:90,1] + 57.220;
   1:  PR[GP1:91,2] = PR[GP1:90,2] + 23.103;
   1:L PR[91] 10mm/sec CNT100;
   1:  PR[GP1:91,1] = PR[GP1:90,1] + 52.715;
   1:  PR[GP1:91,2] = PR[GP1:90,2] + 27.515;
   1:L PR[91] 10mm/sec CNT100;
   1:  PR[GP1:91,1] = PR[GP1:90,1] + 50.419;
   1:  PR[GP1:91,2] = PR[GP1:90,2] + 29.593;
   1:L PR[91] 10mm/sec CNT100;
   1:  PR[GP1:91,1] = PR[GP1:90,1] + 45.137;
   1:  PR[GP1:91,2] = PR[GP1:90,2] + 32.907;
   1:L PR[91] 10mm/sec CNT100;
   1:  PR[GP1:91,1] = PR[GP1:90,1] + 41.674;
   1:  PR[GP1:91,2] = PR[GP1:90,2] + 34.420;
   1:L PR[91] 10mm/sec CNT100;
   1:  PR[GP1:91,1] = PR[GP1:90,1] + 35.930;
   1:  PR[GP1:91,2] = PR[GP1:90,2] + 36.516;
   1:L PR[91] 10mm/sec CNT100;
   1:  PR[GP1:91,1] = PR[GP1:90,1] + 30.492;
   1:  PR[GP1:91,2] = PR[GP1:90,2] + 37.287;
   1:L PR[91] 10mm/sec CNT100;
   1:  PR[GP1:91,1] = PR[GP1:90,1] + 25.611;
   1:  PR[GP1:91,2] = PR[GP1:90,2] + 37.741;
   1:L PR[91] 10mm/sec CNT100;
   1:  PR[GP1:91,1] = PR[GP1:90,1] + 20.398;
   1:  PR[GP1:91,2] = PR[GP1:90,2] + 37.394;
   1:L PR[91] 10mm/sec CNT100;
   1:  PR[GP1:91,1] = PR[GP1:90,1] + 14.853;
   1:  PR[GP1:91,2] = PR[GP1:90,2] + 36.085;
   1:L PR[91] 10mm/sec CNT100;
   1:  PR[GP1:91,1] = PR[GP1:90,1] + 10.109;
   1:  PR[GP1:91,2] = PR[GP1:90,2] + 34.721;
   1:L PR[91] 10mm/sec CNT100;
   1:  PR[GP1:91,1] = PR[GP1:90,1] + 5.724;
   1:  PR[GP1:91,2] = PR[GP1:90,2] + 32.366;
   1:L PR[91] 10mm/sec CNT100;
   1:  PR[GP1:91,1] = PR[GP1:90,1] + -0.263;
   1:  PR[GP1:91,2] = PR[GP1:90,2] + 27.496;
   1:L PR[91] 10mm/sec CNT100;
   1:  PR[GP1:91,1] = PR[GP1:90,1] + -6.234;
   1:  PR[GP1:91,2] = PR[GP1:90,2] + 32.351;
   1:L PR[91] 10mm/sec CNT100;
